// TIA Portal project "Project" (V15)

(* hardware
DEVICE "S7300/ET200M station_2"  S7-300 station
   slot 0: "Rail_0"  Rail  6ES7 390-1***0-0AA0
   slot 2: "PLC_2"  CPU 319-3 PN/DP  6ES7 318-3EL01-0AB0  V3.2
      slot 2: "DP interface_1"  DP
      slot 3: "PROFINET interface_1"  PN-IO
         slot 1: "Port_1"  Port
         slot 2: "Port_2"  Port
   slot 4: "DI 16/DO 16x24VDC/0.5A_1"  DI16/DO16 x 24V / 0.5A  6ES7 323-1BL00-0AA0
   slot 5: "DI 16/DO 16x24VDC/0.5A_2"  DI16/DO16 x 24V / 0.5A  6ES7 323-1BL00-0AA0
   slot 6: "DI 16/DO 16x24VDC/0.5A_3"  DI16/DO16 x 24V / 0.5A  6ES7 323-1BL00-0AA0
   slot 7: "DI 16/DO 16x24VDC/0.5A_4"  DI16/DO16 x 24V / 0.5A  6ES7 323-1BL00-0AA0
   slot 8: "DI 16/DO 16x24VDC/0.5A_5"  DI16/DO16 x 24V / 0.5A  6ES7 323-1BL00-0AA0
   slot 9: "DI 16/DO 16x24VDC/0.5A_6"  DI16/DO16 x 24V / 0.5A  6ES7 323-1BL00-0AA0
   slot 10: "DI 16/DO 16x24VDC/0.5A_7"  DI16/DO16 x 24V / 0.5A  6ES7 323-1BL00-0AA0
   slot 11: "DI 16/DO 16x24VDC/0.5A_8"  DI16/DO16 x 24V / 0.5A  6ES7 323-1BL00-0AA0
*)

// ===== PLC "PLC_2"  CPU 319-3 PN/DP =====

VAR_GLOBAL   // PLC tag table "All_Tags"
   "CCC1" AT %I10.0 : Bool;
   "CCC2" AT %I10.1 : Bool;
   "Tag_1" AT %M5.6 : Bool;
   "Tag_2" AT %M5.7 : Bool;
   "Tag_3" AT %M6.0 : Bool;
   "Tag_4" AT %M6.1 : Bool;
   "Tag_5" AT %M6.2 : Bool;
   "Tag_6" AT %M6.3 : Bool;
   "Tag_7" AT %M6.4 : Bool;
   "Tag_8" AT %M6.5 : Bool;
   "Tag_9" AT %M6.6 : Bool;
END_VAR

VAR_GLOBAL   // PLC tag table "base_feeding_station"
   "lid_detection" AT %I0.0 : Bool;
   "stop_beginning_lid_sensor" AT %I0.1 : Bool;
   "start_LID_feeding_convyer" AT %I0.2 : Bool;
   "LID_detected_grip" AT %I0.3 : Bool;
   "stop_LID_Feeding" AT %I0.4 : Bool;
   "LID_machining_entrance_sensor" AT %I0.5 : Bool;
   "base_Raw_counter_start" AT %I0.6 : Bool;
   "stop_base_begininning_convyr" AT %I0.7 : Bool;
   "base_gripper_detected" AT %I1.0 : Bool;
   "start_base_raw_feeding" AT %I1.1 : Bool;
   "stop_base_raw_feeding" AT %I1.2 : Bool;
   "stop_base_machining_convyr" AT %I1.3 : Bool;
   "lid_start_button" AT %I1.4 : Bool;
   "lid_stop_button" AT %I1.5 : Bool;
   "lid_emergency_button" AT %I1.6 : Bool;
   "base_start_button" AT %I1.7 : Bool;
   "base_stop_button" AT %I2.0 : Bool;
   "base_emergency" AT %I2.1 : Bool;
   "Lid_beginning_conveyr" AT %Q0.0 : Bool;
   "lid_feeding_conveyr" AT %Q0.1 : Bool;
   "Lid_pickup_x_axis" AT %Q0.3 : Bool;
   "lid_pickup_z_axis" AT %Q0.4 : Bool;
   "lid_sucction_gripper" AT %Q0.5 : Bool;
   "base_beginning_conveyr" AT %Q0.6 : Bool;
   "lid-machinning_conveyr" AT %Q0.2 : Bool;
   "base_raw_feeding_conveyr" AT %Q0.7 : Bool;
   "base_to_machinning_conveyr" AT %Q1.0 : Bool;
   "base_pickup_x_axis" AT %Q1.1 : Bool;
   "base_pickup_z_axis" AT %Q1.2 : Bool;
   "base_sucction_gripper" AT %Q1.3 : Bool;
   "base_start_button_1_light" AT %Q1.4 : Bool;
   "base_stop_button_1_light" AT %Q1.5 : Bool;
   "lid_start_light" AT %Q1.6 : Bool;
   "lid_stop_button_1_light" AT %Q1.7 : Bool;
   "base_raw_material" AT %Q2.0 : Bool;
   "lid_raw_emit" AT %Q2.1 : Bool;
   "state_of_start_base" AT %M0.0 : Bool;
   "state_of_start_LID" AT %M0.1 : Bool;
   "state_of_lid" AT %M0.2 : Bool;
   "dummy" AT %M0.3 : Bool;
   "To_emit_lid" AT %M0.4 : Bool;
   "item_ready_to_picked" AT %M0.5 : Bool;
   "movin_lid_z_mem" AT %M0.6 : Bool;
   "LID_moving_z_sensor" AT %I2.4 : Bool;
   "LID_moving_x_sensor" AT %I2.5 : Bool;
   "dummy(1)" AT %M0.7 : Bool;
   "dummy(2)" AT %M1.0 : Bool;
   "lid_belt_convyer_excess" AT %Q2.2 : Bool;
   "push_excess_blue_lid" AT %Q2.3 : Bool;
   "push_excess_green_lid" AT %Q2.4 : Bool;
   "Blue_vision_lid" AT %I2.6 : Bool;
   "green_vision_lid" AT %I2.7 : Bool;
   "front_blue_push_lid" AT %I3.0 : Bool;
   "back_blue_push_lid" AT %I3.1 : Bool;
   "front_green_push_lid" AT %I3.2 : Bool;
   "back_green_push_lid" AT %I3.3 : Bool;
   "into_cnc_lid_sensor" AT %I3.4 : Bool;
   "CNC_lid_empty" AT %M1.1 : Bool;
   "ONE_OBJECT_IN" AT %Q2.5 : Bool;
   "KEEP_DISTANCE" AT %Q2.6 : Bool;
   "ARE_WE_THERE_YET_BLUE_lid" AT %M1.2 : Bool;
   "ARE_WE_THERE_YET_GREEN_lid" AT %M1.3 : Bool;
   "LID_COUNTER_RESET_BUTTON_BLUE" AT %I3.5 : Bool;
   "TO_STORAGE_BLUE_CONVYER_lid" AT %Q2.7 : Bool;
   "TO_STORAGE_GREEN_CONVYER_lid" AT %Q3.0 : Bool;
   "TO_STORAGE_BLUE_SENSOR_lid" AT %I3.6 : Bool;
   "TO_STORAGE_GREEN_SENSOR_lid" AT %I3.7 : Bool;
   "LID_COUNTER_RESET_BUTTON_GREEN" AT %I4.0 : Bool;
   "GREEN_LID_PUSHER_SORTING(FRONT LIMIT)" AT %I4.1 : Bool;
   "GREEN_LID_PUSHER_SORTING(BACK LIMITT)" AT %I4.2 : Bool;
   "BLUE_LID_PUSHER_SORTING(FRONT LIMIT)" AT %I4.3 : Bool;
   "BLUE_LID_PUSHER_SORTING(BACK LIMIT)" AT %I4.4 : Bool;
   "BEGIN_SORTING_STATION_LIDS" AT %I4.5 : Bool;
   "BLUE_LID_VISION_SORTING" AT %I4.6 : Bool;
   "GREEN_LID_VISION_SORTING" AT %I4.7 : Bool;
   "SORTING_CONVYER_LID" AT %Q3.1 : Bool;
   "GREEN_LID_PUSHER_SORTING" AT %Q3.2 : Bool;
   "BLUE_LID_PUSHER_SORTING" AT %Q3.3 : Bool;
   "CNC_base_empty" AT %M2.5 : Bool;
   "to_emit_base" AT %M1.5 : Bool;
   "base_into_cnc" AT %I5.0 : Bool;
   "BASE_MOVE_X_SENSOR" AT %I5.1 : Bool;
   "BASE_MOVE_Z_SENSOR" AT %I5.2 : Bool;
   "DUMMY1" AT %M1.6 : Bool;
   "DUMMY2" AT %M1.7 : Bool;
   "DUMMY3" AT %M2.0 : Bool;
   "DUMMY4" AT %M2.1 : Bool;
   "DUMMY5" AT %M2.2 : Bool;
   "BASE_RAW_EXESS_CONV" AT %Q3.4 : Bool;
   "Are_we_there_base_raw_blue" AT %M2.3 : Bool;
   "Are_we_there_base_raw_green" AT %M2.4 : Bool;
   "base_raw_blue_exes_vision" AT %I5.3 : Bool;
   "base_raw_green_exes_vision" AT %I5.4 : Bool;
   "to_blue_base_raw_storage_sensor" AT %I5.5 : Bool;
   "to_green_base_raw_storage_sensor" AT %I5.6 : Bool;
   "push_ex_green_base raw(front)" AT %I5.7 : Bool;
   "push_ex_green_base raw (back)" AT %I6.0 : Bool;
   "pusher blue base raw (front)" AT %I6.1 : Bool;
   "pusher blue base raw (back)" AT %I6.2 : Bool;
   "is_base_exsist" AT %M1.4 : Bool;
   "Conv_sorting_set_base" AT %M2.6 : Bool;
   "BEGIN_SORTING_STATION_BASE_4" AT %Q5.3 : Bool;
END_VAR

VAR_GLOBAL   // PLC tag table "Assembly_tags"
   "Assembly green lid start" AT %I8.0 : Bool;
   "Assembly blue lid start" AT %I8.1 : Bool;
   "Assembly green base start" AT %I8.2 : Bool;
   "Assembly blue base start" AT %I8.3 : Bool;
   "G_lid in place" AT %I8.4 : Bool;
   "G_base in place" AT %I8.5 : Bool;
   "G_lid_clamped" AT %I8.6 : Bool;
   "G_base_clamped" AT %I8.7 : Bool;
   "G_part_leaving" AT %I9.0 : Bool;
   "G_item_detect" AT %I9.1 : Bool;
   "B_lid in place" AT %I9.2 : Bool;
   "B_base in place" AT %I9.3 : Bool;
   "B_lid_clamped" AT %I9.4 : Bool;
   "B_base_clamped" AT %I9.5 : Bool;
   "B_part_leaving" AT %I9.6 : Bool;
   "B_item_detect" AT %I9.7 : Bool;
   "G_Negative_Trig_1" AT %M4.0 : Bool;
   "G_Negative_Trig_2" AT %M4.1 : Bool;
   "G_Negative_Trig_3" AT %M4.2 : Bool;
   "move_green_lid_conv" AT %M4.3 : Bool;
   "move_green_base_conv" AT %M4.4 : Bool;
   "move_blue_lid_conv" AT %M4.5 : Bool;
   "move_blue_base_conv" AT %M4.6 : Bool;
   "B_Negative_Trig_1" AT %M4.7 : Bool;
   "B_Negative_Trig_2" AT %M5.0 : Bool;
   "B_Negative_Trig_3" AT %M5.1 : Bool;
   "G_Detected_Memory" AT %M5.2 : Bool;
   "G_Reset" AT %M5.3 : Bool;
   "B_Detected_Memory" AT %M5.4 : Bool;
   "B_Reset" AT %M5.5 : Bool;
   "G_Timer_1" AT %T0 : Timer;
   "G_Timer_2" AT %T1 : Timer;
   "G_Timer_3" AT %T2 : Timer;
   "B_Timer_1" AT %T3 : Timer;
   "B_Timer_2" AT %T4 : Timer;
   "B_Timer_3" AT %T5 : Timer;
   "G_lids_conv_1" AT %Q7.0 : Bool;
   "G_lids_conv_2" AT %Q7.1 : Bool;
   "G_lids_conv_3" AT %Q7.2 : Bool;
   "G_lids_conv_4" AT %Q7.3 : Bool;
   "G_lids_conv_5" AT %Q7.4 : Bool;
   "G_lids_conv_6" AT %Q7.5 : Bool;
   "G_lids_conv_7" AT %Q7.6 : Bool;
   "G_lids_conv_8" AT %Q7.7 : Bool;
   "B_lids_conv_1" AT %Q8.0 : Bool;
   "B_lids_conv_2" AT %Q8.1 : Bool;
   "B_lids_conv_3" AT %Q8.2 : Bool;
   "B_lids_conv_4" AT %Q8.3 : Bool;
   "G_base_conv_1" AT %Q8.4 : Bool;
   "G_base_conv_2" AT %Q8.5 : Bool;
   "G_base_conv_3" AT %Q8.6 : Bool;
   "G_base_conv_4" AT %Q8.7 : Bool;
   "G_base_conv_5" AT %Q9.0 : Bool;
   "G_base_conv_6" AT %Q9.1 : Bool;
   "B_base_conv_1" AT %Q9.2 : Bool;
   "B_base_conv_2" AT %Q9.3 : Bool;
   "B_base_conv_3" AT %Q9.4 : Bool;
   "B_base_conv_4" AT %Q9.5 : Bool;
   "G_clamp_lid" AT %Q9.6 : Bool;
   "G_clamp_base" AT %Q9.7 : Bool;
   "G_move Z" AT %Q10.0 : Bool;
   "G_grab" AT %Q10.1 : Bool;
   "G_move X" AT %Q10.2 : Bool;
   "G_pos.Raise_bases" AT %Q10.3 : Bool;
   "B_clamp_lid" AT %Q10.4 : Bool;
   "B_clamp_base" AT %Q10.5 : Bool;
   "B_move Z" AT %Q10.6 : Bool;
   "B_grab" AT %Q10.7 : Bool;
   "B_move X" AT %Q11.0 : Bool;
   "B_pos.Raise_bases" AT %Q11.1 : Bool;
END_VAR

VAR_GLOBAL   // PLC tag table "Default tag table"
   "MachineCenter1_lid_start" AT %Q3.5 : Bool;
   "MachineCenter1_lid_produceLids" AT %Q3.6 : Bool;
   "push_excess_blue_base" AT %Q3.7 : Bool;
   "push_excess_green_base" AT %Q4.0 : Bool;
   "base_COUNTER_RESET_BUTTON_BLUE" AT %I6.3 : Bool;
   "base_COUNTER_RESET_BUTTON_GREEN" AT %I6.4 : Bool;
   "base_raw_excess_blue" AT %Q4.1 : Bool;
   "base_raw_excess_green" AT %Q4.2 : Bool;
   "base_vision_raw_execess_sensor_green" AT %I6.5 : Bool;
   "base_vision_raw_execess_sensor_blue" AT %I6.6 : Bool;
   "MachineCenter2_base_start" AT %Q4.3 : Bool;
   "Stop_blade4" AT %Q4.4 : Bool;
   "Stop_blade5" AT %Q4.5 : Bool;
   "MACHINE1_BUSY" AT %I6.7 : Bool;
   "BEGIN_SORTING_STATION_BASE_SENSOR" AT %I7.0 : Bool;
   "BEGIN_SORTING_STATION_BASE_1" AT %Q4.6 : Bool;
   "BEGIN_SORTING_STATION_BASE_2" AT %Q4.7 : Bool;
   "BEGIN_SORTING_STATION_BASE_3" AT %Q5.0 : Bool;
   "Green_base_sorting_vision" AT %I7.1 : Bool;
   "Blue_base_sorting_vision" AT %I7.2 : Bool;
   "Pusher_green_base (Front Limit)" AT %I7.3 : Bool;
   "Pusher_green_base (Back Limit)" AT %I7.4 : Bool;
   "Pusher_blue_base (Front Limit)" AT %I7.5 : Bool;
   "Pusher_blue_base (Back Limit)" AT %I7.6 : Bool;
   "Pusher_blue_base_sorter" AT %Q5.2 : Bool;
   "Pusher_green_base_sorter" AT %Q5.1 : Bool;
   "Conv_sorting_set_lid" AT %M2.7 : Bool;
   "Emit_set_lid" AT %M3.0 : Bool;
   "Emit_set_base" AT %M3.1 : Bool;
   "Blue count" AT %MW4 : Int;
   "excess blue lid raw led light" AT %Q5.4 : Bool;
   "excess green lid raw led light" AT %Q5.5 : Bool;
   "excess blue base raw led light" AT %Q5.6 : Bool;
   "excess green base raw led light" AT %Q5.7 : Bool;
   "blue lid sorting light" AT %Q6.0 : Bool;
   "green lid sorting light" AT %Q6.1 : Bool;
   "blue base sorting light" AT %Q6.2 : Bool;
   "green base sorting light" AT %Q6.3 : Bool;
   "Green_Lid_conv_timer" AT %T6 : Timer;
   "Blue_Lid_conv_timer" AT %T7 : Timer;
   "Green_Base_conv_timer" AT %T8 : Timer;
   "Blue_Base_conv_timer" AT %T9 : Timer;
END_VAR

DATA_BLOCK "Data_block_1ddd"   // DB3
{ S7_Optimized_Access := 'FALSE' }
VERSION : 0.1
BEGIN
END_DATA_BLOCK

DATA_BLOCK "PICK_UP_LID_ROBOT_DB"   // DB11
{ S7_Optimized_Access := 'FALSE' }
VERSION : 0.1
// stored: InstanceOfName PICK_UP_LID_ROBOT
"PICK_UP_LID_ROBOT"
BEGIN
END_DATA_BLOCK

DATA_BLOCK "LID_SORTING_STATION_DB"   // DB12
{ S7_Optimized_Access := 'FALSE' }
VERSION : 0.1
// stored: InstanceOfName LID_SORTING_STATION
"LID_SORTING_STATION"
BEGIN
END_DATA_BLOCK

DATA_BLOCK "LID PRODUCTION_DB"   // DB13
{ S7_Optimized_Access := 'FALSE' }
VERSION : 0.1
// stored: InstanceOfName LID PRODUCTION
"LID PRODUCTION"
BEGIN
END_DATA_BLOCK

DATA_BLOCK "LID_execess_remove_station_DB"   // DB14
{ S7_Optimized_Access := 'FALSE' }
VERSION : 0.1
// stored: InstanceOfName LID_execess_remove_station
"LID_execess_remove_station"
BEGIN
END_DATA_BLOCK

DATA_BLOCK "base_production_fb_DB"   // DB17
{ S7_Optimized_Access := 'FALSE' }
VERSION : 0.1
// stored: InstanceOfName base_production_fb
"base_production_fb"
BEGIN
END_DATA_BLOCK

DATA_BLOCK "PICK_UP_BASE_ROBOT_DB"   // DB19
{ S7_Optimized_Access := 'FALSE' }
VERSION : 0.1
// stored: InstanceOfName PICK_UP_BASE_ROBOT
"PICK_UP_BASE_ROBOT"
BEGIN
END_DATA_BLOCK

DATA_BLOCK "PICK_UP_BASE_ROBOT_DB_1"   // DB20
{ S7_Optimized_Access := 'FALSE' }
VERSION : 0.1
// stored: InstanceOfName PICK_UP_BASE_ROBOT
"PICK_UP_BASE_ROBOT"
BEGIN
END_DATA_BLOCK

DATA_BLOCK "BASE_execess_remove_station_DB"   // DB26
{ S7_Optimized_Access := 'FALSE' }
VERSION : 0.1
// stored: InstanceOfName BASE_execess_remove_station
"BASE_execess_remove_station"
BEGIN
END_DATA_BLOCK

DATA_BLOCK "A_COUNTER_DB_1"   // DB27
{ S7_Optimized_Access := 'FALSE' }
VERSION : 0.1
// stored: InstanceOfName A_COUNTER
"A_COUNTER"
BEGIN
END_DATA_BLOCK

DATA_BLOCK "BASE_SORTING_STATION_DB"   // DB28
{ S7_Optimized_Access := 'FALSE' }
VERSION : 0.1
// stored: InstanceOfName BASE_SORTING_STATION
"BASE_SORTING_STATION"
BEGIN
END_DATA_BLOCK

DATA_BLOCK "Block_1_DB"   // DB30
{ S7_Optimized_Access := 'FALSE' }
VERSION : 0.1
// stored: InstanceOfName A_COUNTER
"A_COUNTER"
BEGIN
END_DATA_BLOCK

DATA_BLOCK "Assembly_conv_DB"   // DB31
{ S7_Optimized_Access := 'FALSE' }
VERSION : 0.1
// stored: InstanceOfName Assembly_conv
"Assembly_conv"
BEGIN
END_DATA_BLOCK

DATA_BLOCK "Assembly_Blue_DB"   // DB32
{ S7_Optimized_Access := 'FALSE' }
VERSION : 0.1
// stored: InstanceOfName Assembly_Blue
"Assembly_Blue"
BEGIN
END_DATA_BLOCK

DATA_BLOCK "Assembly_Green_DB"   // DB33
{ S7_Optimized_Access := 'FALSE' }
VERSION : 0.1
// stored: InstanceOfName Assembly_Green
"Assembly_Green"
BEGIN
END_DATA_BLOCK

DATA_BLOCK "Assembly_Emergency_DB_1"   // DB34
{ S7_Optimized_Access := 'FALSE' }
VERSION : 0.1
// stored: InstanceOfName Assembly_Emergency
"Assembly_Emergency"
BEGIN
END_DATA_BLOCK

DATA_BLOCK "Assembly_Emergency_DB"   // DB35
{ S7_Optimized_Access := 'FALSE' }
VERSION : 0.1
// stored: InstanceOfName Assembly_Emergency
"Assembly_Emergency"
BEGIN
END_DATA_BLOCK

DATA_BLOCK "A_COUNTER_DB"   // DB36
{ S7_Optimized_Access := 'FALSE' }
VERSION : 0.1
// stored: InstanceOfName A_COUNTER
"A_COUNTER"
BEGIN
END_DATA_BLOCK

FUNCTION_BLOCK "PICK_UP_LID_ROBOT"   // FB1, LAD
{ S7_Optimized_Access := 'FALSE' }
VERSION : 0.1
   VAR_TEMP   // added for the SCL form of the ladder/FBD networks
      _w1 : Bool;
   END_VAR
BEGIN

REGION Network 1: LID_PICKUP_ROBOT_LOWERING_Z_AXIS
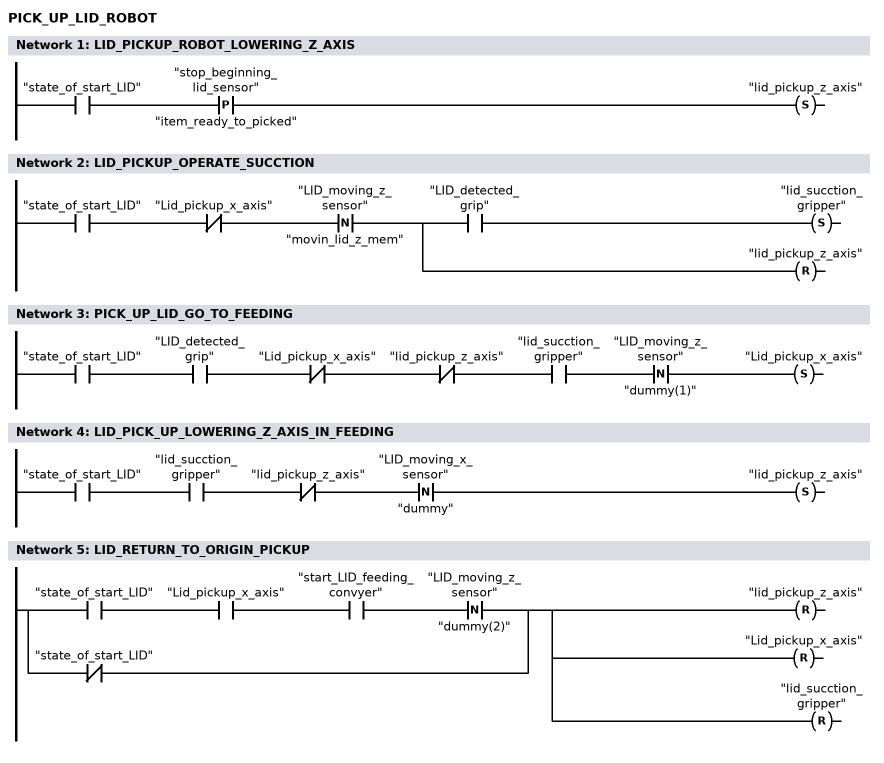
   RUNG wire#powerrail
      Contact( "state_of_start_LID" )
      P_Contact(operand := "stop_beginning_lid_sensor", bit := "item_ready_to_picked")
      S_Coil( "lid_pickup_z_axis" )
   END_RUNG
   // the same network as SCL:
   #_w1 := "state_of_start_LID" AND "stop_beginning_lid_sensor" AND NOT "item_ready_to_picked";   // rising edge of "stop_beginning_lid_sensor"
   "item_ready_to_picked" := "stop_beginning_lid_sensor";
   IF #_w1 THEN "lid_pickup_z_axis" := TRUE; END_IF;
END_REGION

REGION Network 2: LID_PICKUP_OPERATE_SUCCTION
   RUNG wire#powerrail
      Contact( "state_of_start_LID" )
      I_Contact( "Lid_pickup_x_axis" )
      N_Contact(operand := "LID_moving_z_sensor", bit := "movin_lid_z_mem")
      wire#w1
      Contact( "LID_detected_grip" )
      S_Coil( "lid_sucction_gripper" )
   END_RUNG
   RUNG wire#w1
      R_Coil( "lid_pickup_z_axis" )
   END_RUNG
   // the same network as SCL:
   #_w1 := "state_of_start_LID" AND NOT "Lid_pickup_x_axis" AND NOT "LID_moving_z_sensor" AND "movin_lid_z_mem";   // falling edge of "LID_moving_z_sensor"
   "movin_lid_z_mem" := "LID_moving_z_sensor";
   IF #_w1 AND "LID_detected_grip" THEN "lid_sucction_gripper" := TRUE; END_IF;
   IF #_w1 THEN "lid_pickup_z_axis" := FALSE; END_IF;
END_REGION

REGION Network 3: PICK_UP_LID_GO_TO_FEEDING
   RUNG wire#powerrail
      Contact( "state_of_start_LID" )
      Contact( "LID_detected_grip" )
      I_Contact( "Lid_pickup_x_axis" )
      I_Contact( "lid_pickup_z_axis" )
      Contact( "lid_sucction_gripper" )
      N_Contact(operand := "LID_moving_z_sensor", bit := "dummy(1)")
      S_Coil( "Lid_pickup_x_axis" )
   END_RUNG
   // the same network as SCL:
   #_w1 := "state_of_start_LID" AND "LID_detected_grip" AND NOT "Lid_pickup_x_axis" AND NOT "lid_pickup_z_axis" AND "lid_sucction_gripper" AND NOT "LID_moving_z_sensor" AND "dummy(1)";   // falling edge of "LID_moving_z_sensor"
   "dummy(1)" := "LID_moving_z_sensor";
   IF #_w1 THEN "Lid_pickup_x_axis" := TRUE; END_IF;
END_REGION

REGION Network 4: LID_PICK_UP_LOWERING_Z_AXIS_IN_FEEDING
   RUNG wire#powerrail
      Contact( "state_of_start_LID" )
      Contact( "lid_sucction_gripper" )
      I_Contact( "lid_pickup_z_axis" )
      N_Contact(operand := "LID_moving_x_sensor", bit := "dummy")
      S_Coil( "lid_pickup_z_axis" )
   END_RUNG
   // the same network as SCL:
   #_w1 := "state_of_start_LID" AND "lid_sucction_gripper" AND NOT "lid_pickup_z_axis" AND NOT "LID_moving_x_sensor" AND "dummy";   // falling edge of "LID_moving_x_sensor"
   "dummy" := "LID_moving_x_sensor";
   IF #_w1 THEN "lid_pickup_z_axis" := TRUE; END_IF;
END_REGION

REGION Network 5: LID_RETURN_TO_ORIGIN_PICKUP
   RUNG wire#powerrail
      Contact( "state_of_start_LID" )
      Contact( "Lid_pickup_x_axis" )
      Contact( "start_LID_feeding_convyer" )
      N_Contact(operand := "LID_moving_z_sensor", bit := "dummy(2)")
      wire#w1
      R_Coil( "lid_pickup_z_axis" )
   END_RUNG
   RUNG wire#powerrail
      I_Contact( "state_of_start_LID" )
   END_RUNG wire#w1
   RUNG wire#w1
      R_Coil( "Lid_pickup_x_axis" )
   END_RUNG
   RUNG wire#w1
      R_Coil( "lid_sucction_gripper" )
   END_RUNG
   // the same network as SCL:
   #_w1 := "state_of_start_LID" AND "Lid_pickup_x_axis" AND "start_LID_feeding_convyer" AND NOT "LID_moving_z_sensor" AND "dummy(2)";   // falling edge of "LID_moving_z_sensor"
   "dummy(2)" := "LID_moving_z_sensor";
   IF #_w1 OR NOT "state_of_start_LID" THEN
       "lid_pickup_z_axis" := FALSE;
       "Lid_pickup_x_axis" := FALSE;
       "lid_sucction_gripper" := FALSE;
   END_IF;
END_REGION
END_FUNCTION_BLOCK

FUNCTION_BLOCK "LID PRODUCTION"   // FB2, LAD
{ S7_Optimized_Access := 'FALSE' }
VERSION : 0.1
BEGIN

REGION Network 1: LID STARTING HANDLE
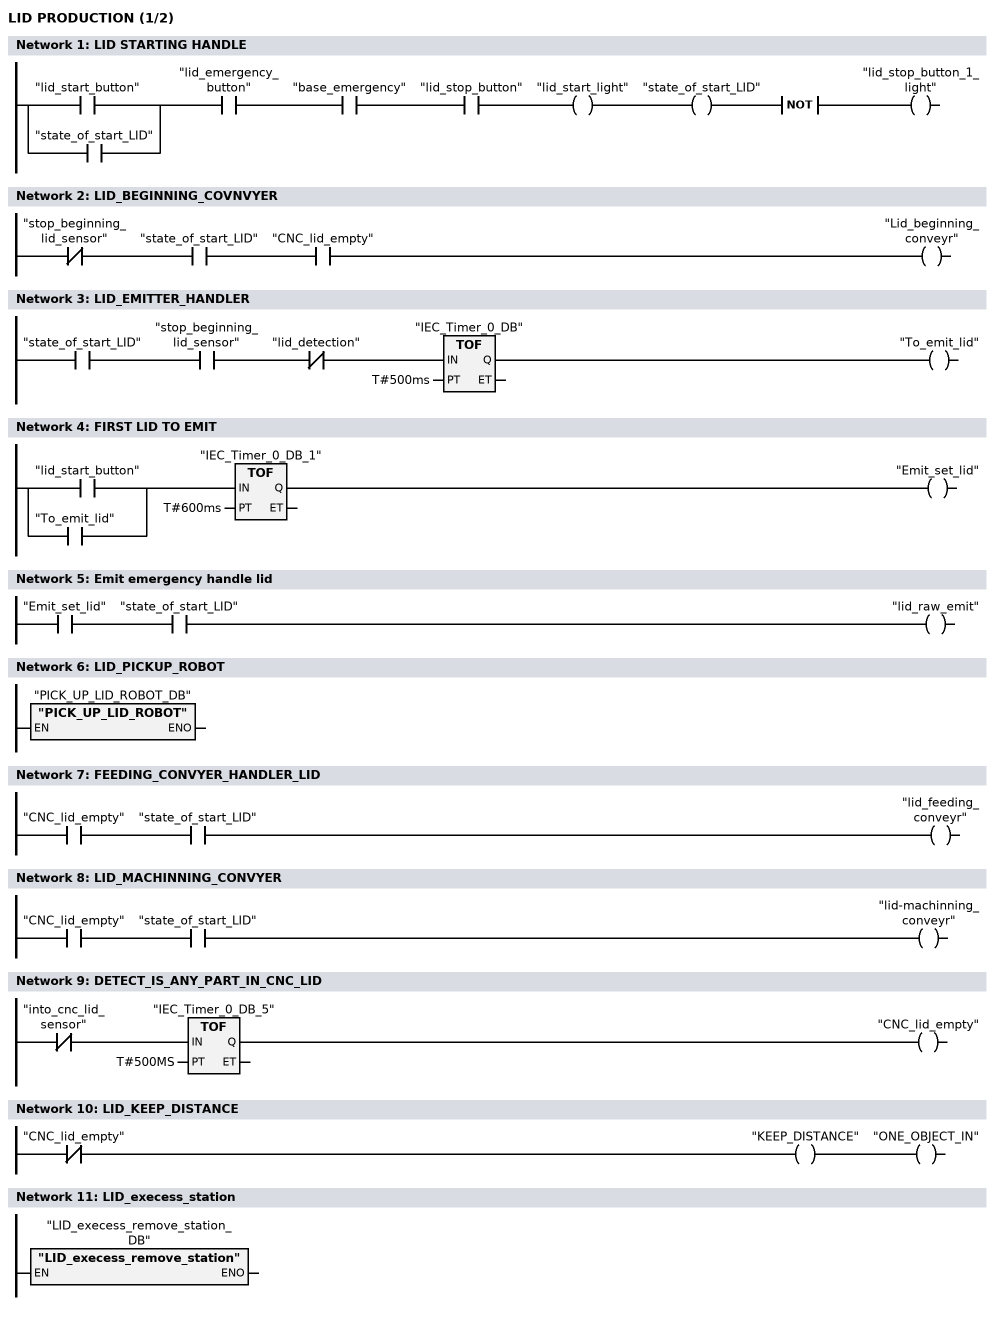
   RUNG wire#powerrail
      Contact( "lid_start_button" )
      wire#w1
      Contact( "lid_emergency_button" )
      Contact( "base_emergency" )
      Contact( "lid_stop_button" )
      Coil( "lid_start_light" )
      Coil( "state_of_start_LID" )
      Not()
      Coil( "lid_stop_button_1_light" )
   END_RUNG
   RUNG wire#powerrail
      Contact( "state_of_start_LID" )
   END_RUNG wire#w1
   // the same network as SCL:
   "lid_start_light" := ("lid_start_button" OR "state_of_start_LID") AND "lid_emergency_button" AND "base_emergency" AND "lid_stop_button";
   "state_of_start_LID" := "lid_start_light";
   "lid_stop_button_1_light" := NOT "lid_start_light";
END_REGION

REGION Network 2: LID_BEGINNING_COVNVYER
   RUNG wire#powerrail
      I_Contact( "stop_beginning_lid_sensor" )
      Contact( "state_of_start_LID" )
      Contact( "CNC_lid_empty" )
      Coil( "Lid_beginning_conveyr" )
   END_RUNG
   // the same network as SCL:
   "Lid_beginning_conveyr" := NOT "stop_beginning_lid_sensor" AND "state_of_start_LID" AND "CNC_lid_empty";
END_REGION

REGION Network 3: LID_EMITTER_HANDLER
   "IEC_Timer_0_DB".TOF(IN := "state_of_start_LID" AND "stop_beginning_lid_sensor" AND NOT "lid_detection",
                        PT := T#500ms);
   "To_emit_lid" := "IEC_Timer_0_DB".Q;
END_REGION

REGION Network 4: FIRST LID TO EMIT
   "IEC_Timer_0_DB_1".TOF(IN := "lid_start_button" OR "To_emit_lid", PT := T#600ms);
   "Emit_set_lid" := "IEC_Timer_0_DB_1".Q;
END_REGION

REGION Network 5: Emit emergency handle lid
   RUNG wire#powerrail
      Contact( "Emit_set_lid" )
      Contact( "state_of_start_LID" )
      Coil( "lid_raw_emit" )
   END_RUNG
   // the same network as SCL:
   "lid_raw_emit" := "Emit_set_lid" AND "state_of_start_LID";
END_REGION

REGION Network 6: LID_PICKUP_ROBOT
   RUNG wire#powerrail
      "PICK_UP_LID_ROBOT_DB"()
   END_RUNG
   // the same network as SCL:
   "PICK_UP_LID_ROBOT_DB"();   // "PICK_UP_LID_ROBOT"
END_REGION

REGION Network 7: FEEDING_CONVYER_HANDLER_LID
   RUNG wire#powerrail
      Contact( "CNC_lid_empty" )
      Contact( "state_of_start_LID" )
      Coil( "lid_feeding_conveyr" )
   END_RUNG
   // the same network as SCL:
   "lid_feeding_conveyr" := "CNC_lid_empty" AND "state_of_start_LID";
END_REGION

REGION Network 8: LID_MACHINNING_CONVYER
   RUNG wire#powerrail
      Contact( "CNC_lid_empty" )
      Contact( "state_of_start_LID" )
      Coil( "lid-machinning_conveyr" )
   END_RUNG
   // the same network as SCL:
   "lid-machinning_conveyr" := "CNC_lid_empty" AND "state_of_start_LID";
END_REGION

REGION Network 9: DETECT_IS_ANY_PART_IN_CNC_LID
   "IEC_Timer_0_DB_5".TOF(IN := NOT "into_cnc_lid_sensor", PT := T#500MS);
   "CNC_lid_empty" := "IEC_Timer_0_DB_5".Q;
END_REGION

REGION Network 10: LID_KEEP_DISTANCE
   RUNG wire#powerrail
      I_Contact( "CNC_lid_empty" )
      Coil( "KEEP_DISTANCE" )
      Coil( "ONE_OBJECT_IN" )
   END_RUNG
   // the same network as SCL:
   "KEEP_DISTANCE" := NOT "CNC_lid_empty";
   "ONE_OBJECT_IN" := NOT "CNC_lid_empty";
END_REGION

REGION Network 11: LID_execess_station
   RUNG wire#powerrail
      "LID_execess_remove_station_DB"()
   END_RUNG
   // the same network as SCL:
   "LID_execess_remove_station_DB"();   // "LID_execess_remove_station"
END_REGION

REGION Network 12: CNC
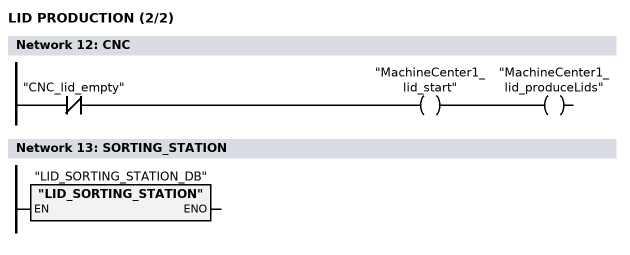
   RUNG wire#powerrail
      I_Contact( "CNC_lid_empty" )
      Coil( "MachineCenter1_lid_start" )
      Coil( "MachineCenter1_lid_produceLids" )
   END_RUNG
   // the same network as SCL:
   "MachineCenter1_lid_start" := NOT "CNC_lid_empty";
   "MachineCenter1_lid_produceLids" := NOT "CNC_lid_empty";
END_REGION

REGION Network 13: SORTING_STATION
   RUNG wire#powerrail
      "LID_SORTING_STATION_DB"()
   END_RUNG
   // the same network as SCL:
   "LID_SORTING_STATION_DB"();   // "LID_SORTING_STATION"
END_REGION
END_FUNCTION_BLOCK

FUNCTION_BLOCK "LID_SORTING_STATION"   // FB3, LAD
{ S7_Optimized_Access := 'FALSE' }
VERSION : 0.1
BEGIN

REGION Network 1: BEGIN SORTING CONVYER
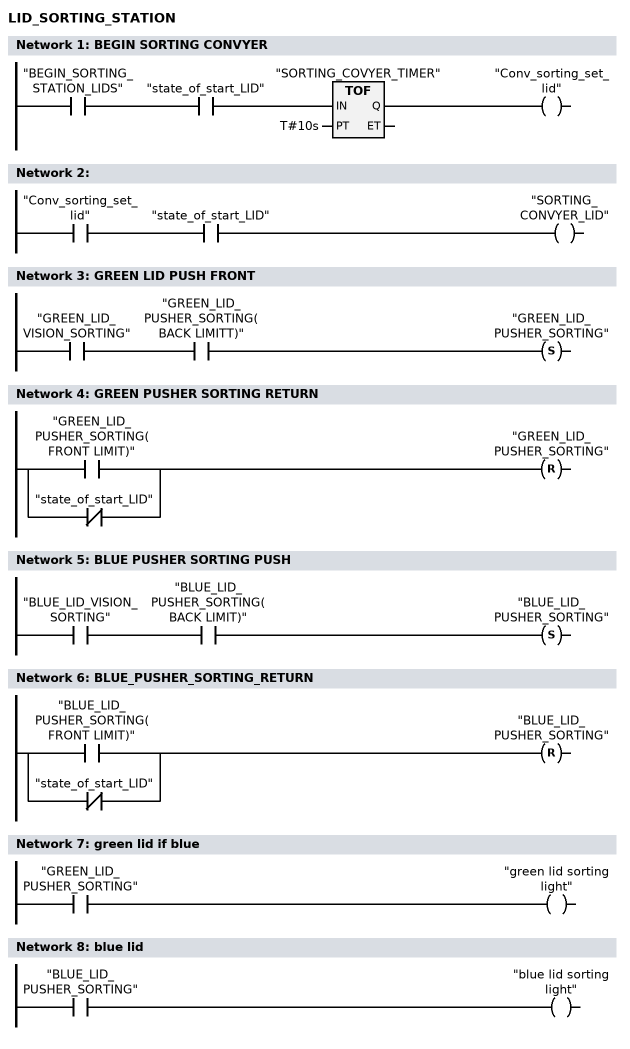
   "SORTING_COVYER_TIMER".TOF(IN := "BEGIN_SORTING_STATION_LIDS" AND "state_of_start_LID", PT := T#10s);
   "Conv_sorting_set_lid" := "SORTING_COVYER_TIMER".Q;
END_REGION

REGION Network 2
   RUNG wire#powerrail
      Contact( "Conv_sorting_set_lid" )
      Contact( "state_of_start_LID" )
      Coil( "SORTING_CONVYER_LID" )
   END_RUNG
   // the same network as SCL:
   "SORTING_CONVYER_LID" := "Conv_sorting_set_lid" AND "state_of_start_LID";
END_REGION

REGION Network 3: GREEN LID PUSH FRONT
   RUNG wire#powerrail
      Contact( "GREEN_LID_VISION_SORTING" )
      Contact( "GREEN_LID_PUSHER_SORTING(BACK LIMITT)" )
      S_Coil( "GREEN_LID_PUSHER_SORTING" )
   END_RUNG
   // the same network as SCL:
   IF "GREEN_LID_VISION_SORTING" AND "GREEN_LID_PUSHER_SORTING(BACK LIMITT)" THEN
       "GREEN_LID_PUSHER_SORTING" := TRUE;
   END_IF;
END_REGION

REGION Network 4: GREEN PUSHER SORTING RETURN
   RUNG wire#powerrail
      Contact( "GREEN_LID_PUSHER_SORTING(FRONT LIMIT)" )
      wire#w1
      R_Coil( "GREEN_LID_PUSHER_SORTING" )
   END_RUNG
   RUNG wire#powerrail
      I_Contact( "state_of_start_LID" )
   END_RUNG wire#w1
   // the same network as SCL:
   IF "GREEN_LID_PUSHER_SORTING(FRONT LIMIT)" OR NOT "state_of_start_LID" THEN
       "GREEN_LID_PUSHER_SORTING" := FALSE;
   END_IF;
END_REGION

REGION Network 5: BLUE PUSHER SORTING PUSH
   RUNG wire#powerrail
      Contact( "BLUE_LID_VISION_SORTING" )
      Contact( "BLUE_LID_PUSHER_SORTING(BACK LIMIT)" )
      S_Coil( "BLUE_LID_PUSHER_SORTING" )
   END_RUNG
   // the same network as SCL:
   IF "BLUE_LID_VISION_SORTING" AND "BLUE_LID_PUSHER_SORTING(BACK LIMIT)" THEN
       "BLUE_LID_PUSHER_SORTING" := TRUE;
   END_IF;
END_REGION

REGION Network 6: BLUE_PUSHER_SORTING_RETURN
   RUNG wire#powerrail
      Contact( "BLUE_LID_PUSHER_SORTING(FRONT LIMIT)" )
      wire#w1
      R_Coil( "BLUE_LID_PUSHER_SORTING" )
   END_RUNG
   RUNG wire#powerrail
      I_Contact( "state_of_start_LID" )
   END_RUNG wire#w1
   // the same network as SCL:
   IF "BLUE_LID_PUSHER_SORTING(FRONT LIMIT)" OR NOT "state_of_start_LID" THEN
       "BLUE_LID_PUSHER_SORTING" := FALSE;
   END_IF;
END_REGION

REGION Network 7: green lid if blue
   RUNG wire#powerrail
      Contact( "GREEN_LID_PUSHER_SORTING" )
      Coil( "green lid sorting light" )
   END_RUNG
   // the same network as SCL:
   "green lid sorting light" := "GREEN_LID_PUSHER_SORTING";
END_REGION

REGION Network 8: blue lid
   RUNG wire#powerrail
      Contact( "BLUE_LID_PUSHER_SORTING" )
      Coil( "blue lid sorting light" )
   END_RUNG
   // the same network as SCL:
   "blue lid sorting light" := "BLUE_LID_PUSHER_SORTING";
END_REGION
END_FUNCTION_BLOCK

FUNCTION_BLOCK "LID_execess_remove_station"   // FB4, LAD
{ S7_Optimized_Access := 'FALSE' }
VERSION : 0.1
   VAR_TEMP   // added for the SCL form of the ladder/FBD networks
      _w1 : Bool;
   END_VAR
BEGIN

REGION Network 1: LID_BELT_EXECESS_CONVYR_HANDLER
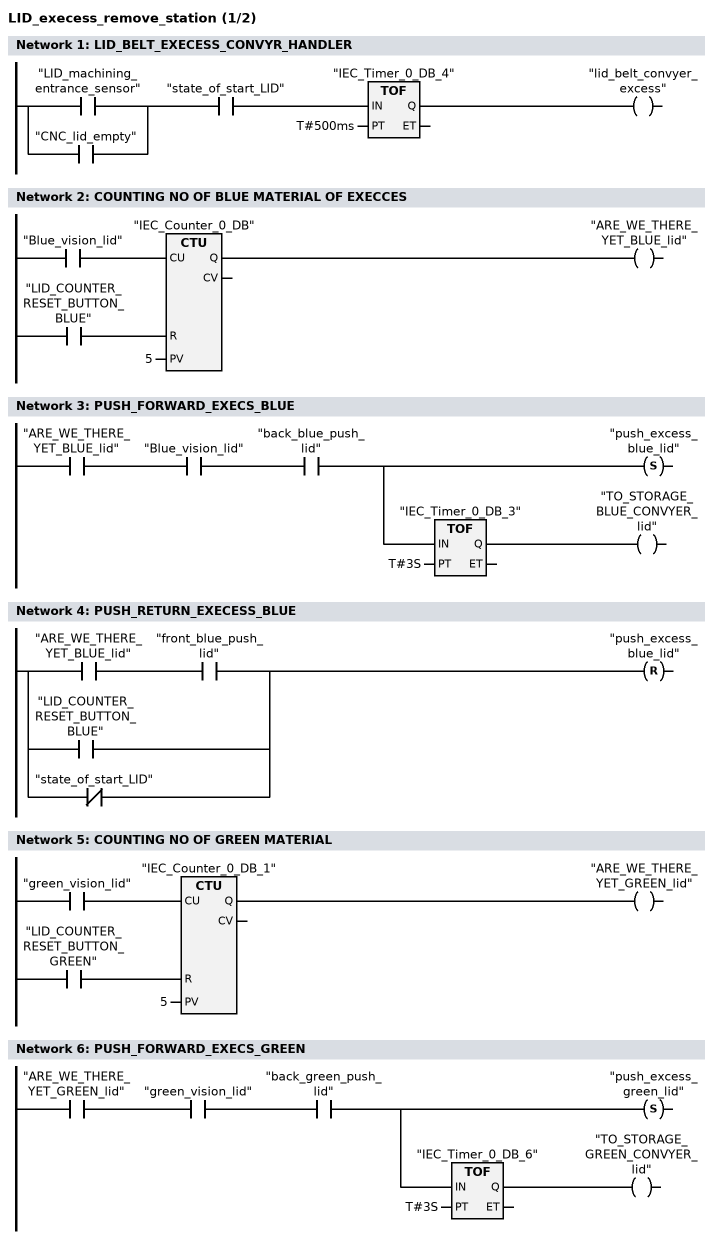
   "IEC_Timer_0_DB_4".TOF(IN := ("LID_machining_entrance_sensor" OR "CNC_lid_empty") AND "state_of_start_LID",
                          PT := T#500ms);
   "lid_belt_convyer_excess" := "IEC_Timer_0_DB_4".Q;
END_REGION

REGION Network 2: COUNTING NO OF BLUE MATERIAL OF EXECCES
   "IEC_Counter_0_DB".CTU(CU := "Blue_vision_lid", R := "LID_COUNTER_RESET_BUTTON_BLUE", PV := 5);
   "ARE_WE_THERE_YET_BLUE_lid" := "IEC_Counter_0_DB".Q;
END_REGION

REGION Network 3: PUSH_FORWARD_EXECS_BLUE
   #_w1 := "ARE_WE_THERE_YET_BLUE_lid" AND "Blue_vision_lid" AND "back_blue_push_lid";
   IF #_w1 THEN "push_excess_blue_lid" := TRUE; END_IF;
   "IEC_Timer_0_DB_3".TOF(IN := #_w1, PT := T#3S);
   "TO_STORAGE_BLUE_CONVYER_lid" := "IEC_Timer_0_DB_3".Q;
END_REGION

REGION Network 4: PUSH_RETURN_EXECESS_BLUE
   RUNG wire#powerrail
      Contact( "ARE_WE_THERE_YET_BLUE_lid" )
      Contact( "front_blue_push_lid" )
      wire#w1
      R_Coil( "push_excess_blue_lid" )
   END_RUNG
   RUNG wire#powerrail
      Contact( "LID_COUNTER_RESET_BUTTON_BLUE" )
   END_RUNG wire#w1
   RUNG wire#powerrail
      I_Contact( "state_of_start_LID" )
   END_RUNG wire#w1
   // the same network as SCL:
   IF ("ARE_WE_THERE_YET_BLUE_lid" AND "front_blue_push_lid") OR "LID_COUNTER_RESET_BUTTON_BLUE" OR NOT "state_of_start_LID" THEN
       "push_excess_blue_lid" := FALSE;
   END_IF;
END_REGION

REGION Network 5: COUNTING NO OF GREEN MATERIAL
   "IEC_Counter_0_DB_1".CTU(CU := "green_vision_lid", R := "LID_COUNTER_RESET_BUTTON_GREEN", PV := 5);
   "ARE_WE_THERE_YET_GREEN_lid" := "IEC_Counter_0_DB_1".Q;
END_REGION

REGION Network 6: PUSH_FORWARD_EXECS_GREEN
   #_w1 := "ARE_WE_THERE_YET_GREEN_lid" AND "green_vision_lid" AND "back_green_push_lid";
   IF #_w1 THEN "push_excess_green_lid" := TRUE; END_IF;
   "IEC_Timer_0_DB_6".TOF(IN := #_w1, PT := T#3S);
   "TO_STORAGE_GREEN_CONVYER_lid" := "IEC_Timer_0_DB_6".Q;
END_REGION

REGION Network 7: PUSH_RETURN_GREEN
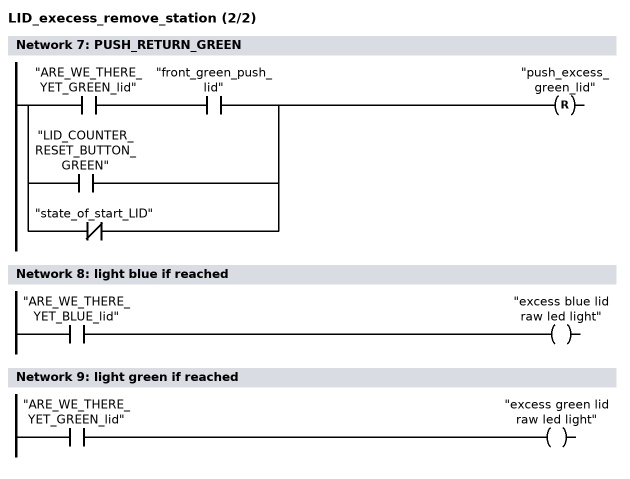
   RUNG wire#powerrail
      Contact( "ARE_WE_THERE_YET_GREEN_lid" )
      Contact( "front_green_push_lid" )
      wire#w1
      R_Coil( "push_excess_green_lid" )
   END_RUNG
   RUNG wire#powerrail
      Contact( "LID_COUNTER_RESET_BUTTON_GREEN" )
   END_RUNG wire#w1
   RUNG wire#powerrail
      I_Contact( "state_of_start_LID" )
   END_RUNG wire#w1
   // the same network as SCL:
   IF ("ARE_WE_THERE_YET_GREEN_lid" AND "front_green_push_lid") OR "LID_COUNTER_RESET_BUTTON_GREEN" OR NOT "state_of_start_LID" THEN
       "push_excess_green_lid" := FALSE;
   END_IF;
END_REGION

REGION Network 8: light blue if reached
   RUNG wire#powerrail
      Contact( "ARE_WE_THERE_YET_BLUE_lid" )
      Coil( "excess blue lid raw led light" )
   END_RUNG
   // the same network as SCL:
   "excess blue lid raw led light" := "ARE_WE_THERE_YET_BLUE_lid";
END_REGION

REGION Network 9: light green if reached
   RUNG wire#powerrail
      Contact( "ARE_WE_THERE_YET_GREEN_lid" )
      Coil( "excess green lid raw led light" )
   END_RUNG
   // the same network as SCL:
   "excess green lid raw led light" := "ARE_WE_THERE_YET_GREEN_lid";
END_REGION
END_FUNCTION_BLOCK

FUNCTION_BLOCK "base_production_fb"   // FB5, LAD
{ S7_Optimized_Access := 'FALSE' }
VERSION : 0.1
BEGIN

REGION Network 1: base_production_station
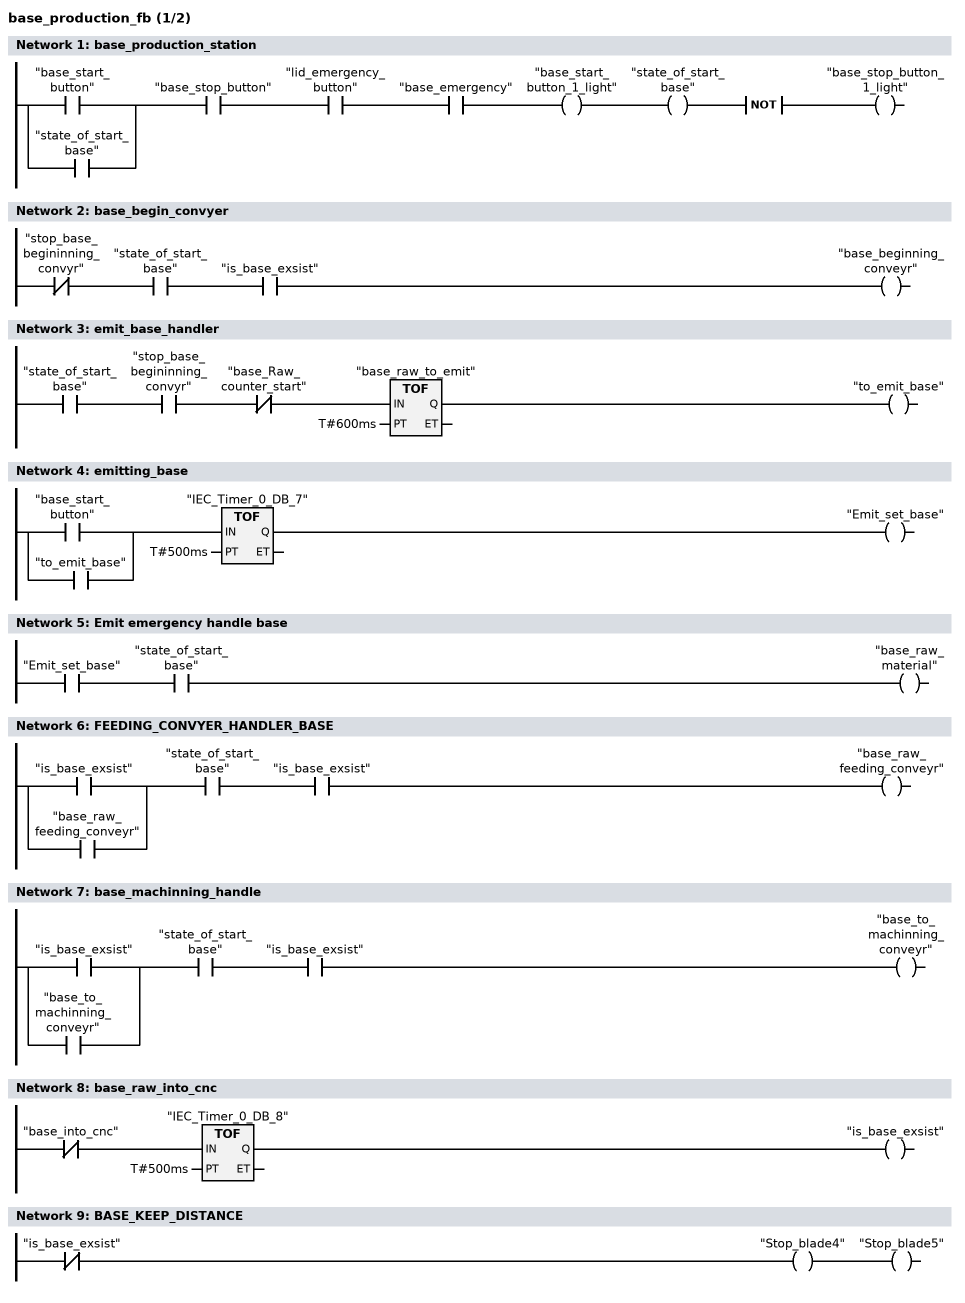
   RUNG wire#powerrail
      Contact( "base_start_button" )
      wire#w1
      Contact( "base_stop_button" )
      Contact( "lid_emergency_button" )
      Contact( "base_emergency" )
      Coil( "base_start_button_1_light" )
      Coil( "state_of_start_base" )
      Not()
      Coil( "base_stop_button_1_light" )
   END_RUNG
   RUNG wire#powerrail
      Contact( "state_of_start_base" )
   END_RUNG wire#w1
   // the same network as SCL:
   "base_start_button_1_light" := ("base_start_button" OR "state_of_start_base") AND "base_stop_button" AND "lid_emergency_button" AND "base_emergency";
   "state_of_start_base" := "base_start_button_1_light";
   "base_stop_button_1_light" := NOT "base_start_button_1_light";
END_REGION

REGION Network 2: base_begin_convyer
   RUNG wire#powerrail
      I_Contact( "stop_base_begininning_convyr" )
      Contact( "state_of_start_base" )
      Contact( "is_base_exsist" )
      Coil( "base_beginning_conveyr" )
   END_RUNG
   // the same network as SCL:
   "base_beginning_conveyr" := NOT "stop_base_begininning_convyr" AND "state_of_start_base" AND "is_base_exsist";
END_REGION

REGION Network 3: emit_base_handler
   "base_raw_to_emit".TOF(IN := "state_of_start_base" AND "stop_base_begininning_convyr" AND NOT "base_Raw_counter_start",
                          PT := T#600ms);
   "to_emit_base" := "base_raw_to_emit".Q;
END_REGION

REGION Network 4: emitting_base
   "IEC_Timer_0_DB_7".TOF(IN := "base_start_button" OR "to_emit_base", PT := T#500ms);
   "Emit_set_base" := "IEC_Timer_0_DB_7".Q;
END_REGION

REGION Network 5: Emit emergency handle base
   RUNG wire#powerrail
      Contact( "Emit_set_base" )
      Contact( "state_of_start_base" )
      Coil( "base_raw_material" )
   END_RUNG
   // the same network as SCL:
   "base_raw_material" := "Emit_set_base" AND "state_of_start_base";
END_REGION

REGION Network 6: FEEDING_CONVYER_HANDLER_BASE
   RUNG wire#powerrail
      Contact( "is_base_exsist" )
      wire#w1
      Contact( "state_of_start_base" )
      Contact( "is_base_exsist" )
      Coil( "base_raw_feeding_conveyr" )
   END_RUNG
   RUNG wire#powerrail
      Contact( "base_raw_feeding_conveyr" )
   END_RUNG wire#w1
   // the same network as SCL:
   "base_raw_feeding_conveyr" := ("is_base_exsist" OR "base_raw_feeding_conveyr") AND "state_of_start_base" AND "is_base_exsist";
END_REGION

REGION Network 7: base_machinning_handle
   RUNG wire#powerrail
      Contact( "is_base_exsist" )
      wire#w1
      Contact( "state_of_start_base" )
      Contact( "is_base_exsist" )
      Coil( "base_to_machinning_conveyr" )
   END_RUNG
   RUNG wire#powerrail
      Contact( "base_to_machinning_conveyr" )
   END_RUNG wire#w1
   // the same network as SCL:
   "base_to_machinning_conveyr" := ("is_base_exsist" OR "base_to_machinning_conveyr") AND "state_of_start_base" AND "is_base_exsist";
END_REGION

REGION Network 8: base_raw_into_cnc
   "IEC_Timer_0_DB_8".TOF(IN := NOT "base_into_cnc", PT := T#500ms);
   "is_base_exsist" := "IEC_Timer_0_DB_8".Q;
END_REGION

REGION Network 9: BASE_KEEP_DISTANCE
   RUNG wire#powerrail
      I_Contact( "is_base_exsist" )
      Coil( "Stop_blade4" )
      Coil( "Stop_blade5" )
   END_RUNG
   // the same network as SCL:
   "Stop_blade4" := NOT "is_base_exsist";
   "Stop_blade5" := NOT "is_base_exsist";
END_REGION

REGION Network 10: base_excess
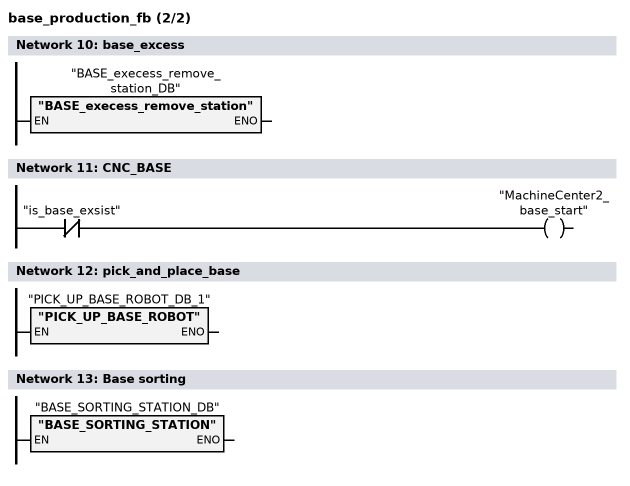
   RUNG wire#powerrail
      "BASE_execess_remove_station_DB"()
   END_RUNG
   // the same network as SCL:
   "BASE_execess_remove_station_DB"();   // "BASE_execess_remove_station"
END_REGION

REGION Network 11: CNC_BASE
   RUNG wire#powerrail
      I_Contact( "is_base_exsist" )
      Coil( "MachineCenter2_base_start" )
   END_RUNG
   // the same network as SCL:
   "MachineCenter2_base_start" := NOT "is_base_exsist";
END_REGION

REGION Network 12: pick_and_place_base
   RUNG wire#powerrail
      "PICK_UP_BASE_ROBOT_DB_1"()
   END_RUNG
   // the same network as SCL:
   "PICK_UP_BASE_ROBOT_DB_1"();   // "PICK_UP_BASE_ROBOT"
END_REGION

REGION Network 13: Base sorting
   RUNG wire#powerrail
      "BASE_SORTING_STATION_DB"()
   END_RUNG
   // the same network as SCL:
   "BASE_SORTING_STATION_DB"();   // "BASE_SORTING_STATION"
END_REGION
END_FUNCTION_BLOCK

FUNCTION_BLOCK "PICK_UP_BASE_ROBOT"   // FB6, LAD
{ S7_Optimized_Access := 'FALSE' }
VERSION : 0.1
   VAR_TEMP   // added for the SCL form of the ladder/FBD networks
      _w1 : Bool;
   END_VAR
BEGIN

REGION Network 1: BASE_PICKUP_ROBOT_LOWERING_Z_AXIS
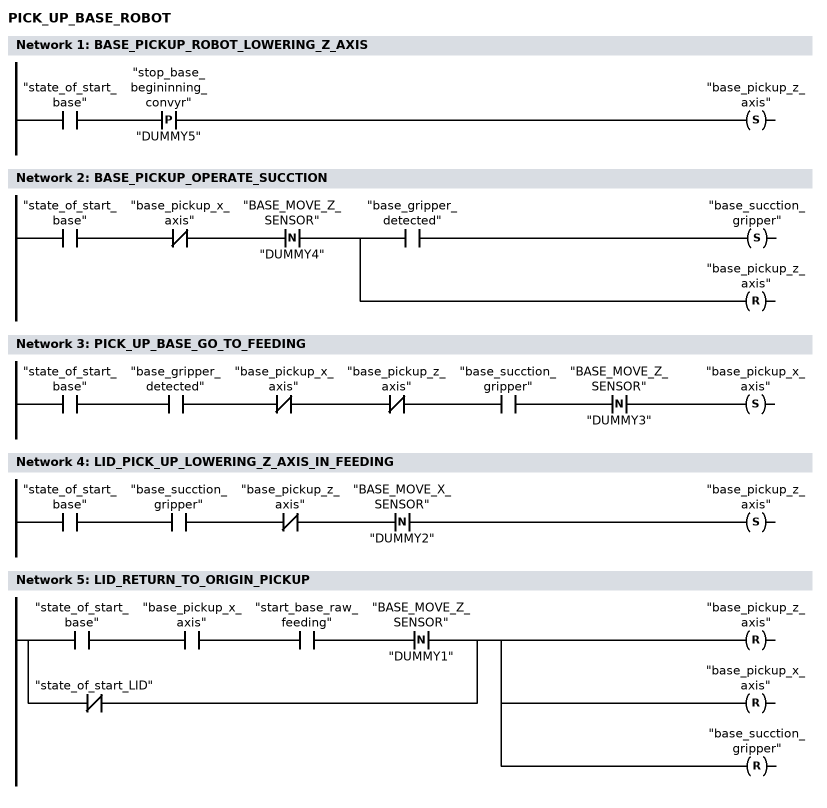
   RUNG wire#powerrail
      Contact( "state_of_start_base" )
      P_Contact(operand := "stop_base_begininning_convyr", bit := "DUMMY5")
      S_Coil( "base_pickup_z_axis" )
   END_RUNG
   // the same network as SCL:
   #_w1 := "state_of_start_base" AND "stop_base_begininning_convyr" AND NOT "DUMMY5";   // rising edge of "stop_base_begininning_convyr"
   "DUMMY5" := "stop_base_begininning_convyr";
   IF #_w1 THEN "base_pickup_z_axis" := TRUE; END_IF;
END_REGION

REGION Network 2: BASE_PICKUP_OPERATE_SUCCTION
   RUNG wire#powerrail
      Contact( "state_of_start_base" )
      I_Contact( "base_pickup_x_axis" )
      N_Contact(operand := "BASE_MOVE_Z_SENSOR", bit := "DUMMY4")
      wire#w1
      Contact( "base_gripper_detected" )
      S_Coil( "base_sucction_gripper" )
   END_RUNG
   RUNG wire#w1
      R_Coil( "base_pickup_z_axis" )
   END_RUNG
   // the same network as SCL:
   #_w1 := "state_of_start_base" AND NOT "base_pickup_x_axis" AND NOT "BASE_MOVE_Z_SENSOR" AND "DUMMY4";   // falling edge of "BASE_MOVE_Z_SENSOR"
   "DUMMY4" := "BASE_MOVE_Z_SENSOR";
   IF #_w1 AND "base_gripper_detected" THEN "base_sucction_gripper" := TRUE; END_IF;
   IF #_w1 THEN "base_pickup_z_axis" := FALSE; END_IF;
END_REGION

REGION Network 3: PICK_UP_BASE_GO_TO_FEEDING
   RUNG wire#powerrail
      Contact( "state_of_start_base" )
      Contact( "base_gripper_detected" )
      I_Contact( "base_pickup_x_axis" )
      I_Contact( "base_pickup_z_axis" )
      Contact( "base_sucction_gripper" )
      N_Contact(operand := "BASE_MOVE_Z_SENSOR", bit := "DUMMY3")
      S_Coil( "base_pickup_x_axis" )
   END_RUNG
   // the same network as SCL:
   #_w1 := "state_of_start_base" AND "base_gripper_detected" AND NOT "base_pickup_x_axis" AND NOT "base_pickup_z_axis" AND "base_sucction_gripper" AND NOT "BASE_MOVE_Z_SENSOR" AND "DUMMY3";   // falling edge of "BASE_MOVE_Z_SENSOR"
   "DUMMY3" := "BASE_MOVE_Z_SENSOR";
   IF #_w1 THEN "base_pickup_x_axis" := TRUE; END_IF;
END_REGION

REGION Network 4: LID_PICK_UP_LOWERING_Z_AXIS_IN_FEEDING
   RUNG wire#powerrail
      Contact( "state_of_start_base" )
      Contact( "base_sucction_gripper" )
      I_Contact( "base_pickup_z_axis" )
      N_Contact(operand := "BASE_MOVE_X_SENSOR", bit := "DUMMY2")
      S_Coil( "base_pickup_z_axis" )
   END_RUNG
   // the same network as SCL:
   #_w1 := "state_of_start_base" AND "base_sucction_gripper" AND NOT "base_pickup_z_axis" AND NOT "BASE_MOVE_X_SENSOR" AND "DUMMY2";   // falling edge of "BASE_MOVE_X_SENSOR"
   "DUMMY2" := "BASE_MOVE_X_SENSOR";
   IF #_w1 THEN "base_pickup_z_axis" := TRUE; END_IF;
END_REGION

REGION Network 5: LID_RETURN_TO_ORIGIN_PICKUP
   RUNG wire#powerrail
      Contact( "state_of_start_base" )
      Contact( "base_pickup_x_axis" )
      Contact( "start_base_raw_feeding" )
      N_Contact(operand := "BASE_MOVE_Z_SENSOR", bit := "DUMMY1")
      wire#w1
      R_Coil( "base_pickup_z_axis" )
   END_RUNG
   RUNG wire#powerrail
      I_Contact( "state_of_start_LID" )
   END_RUNG wire#w1
   RUNG wire#w1
      R_Coil( "base_pickup_x_axis" )
   END_RUNG
   RUNG wire#w1
      R_Coil( "base_sucction_gripper" )
   END_RUNG
   // the same network as SCL:
   #_w1 := "state_of_start_base" AND "base_pickup_x_axis" AND "start_base_raw_feeding" AND NOT "BASE_MOVE_Z_SENSOR" AND "DUMMY1";   // falling edge of "BASE_MOVE_Z_SENSOR"
   "DUMMY1" := "BASE_MOVE_Z_SENSOR";
   IF #_w1 OR NOT "state_of_start_LID" THEN
       "base_pickup_z_axis" := FALSE;
       "base_pickup_x_axis" := FALSE;
       "base_sucction_gripper" := FALSE;
   END_IF;
END_REGION
END_FUNCTION_BLOCK

FUNCTION_BLOCK "BASE_execess_remove_station"   // FB7, LAD
{ S7_Optimized_Access := 'FALSE' }
VERSION : 0.1
BEGIN

REGION Network 1: LID_BELT_EXECESS_CONVYR_HANDLER
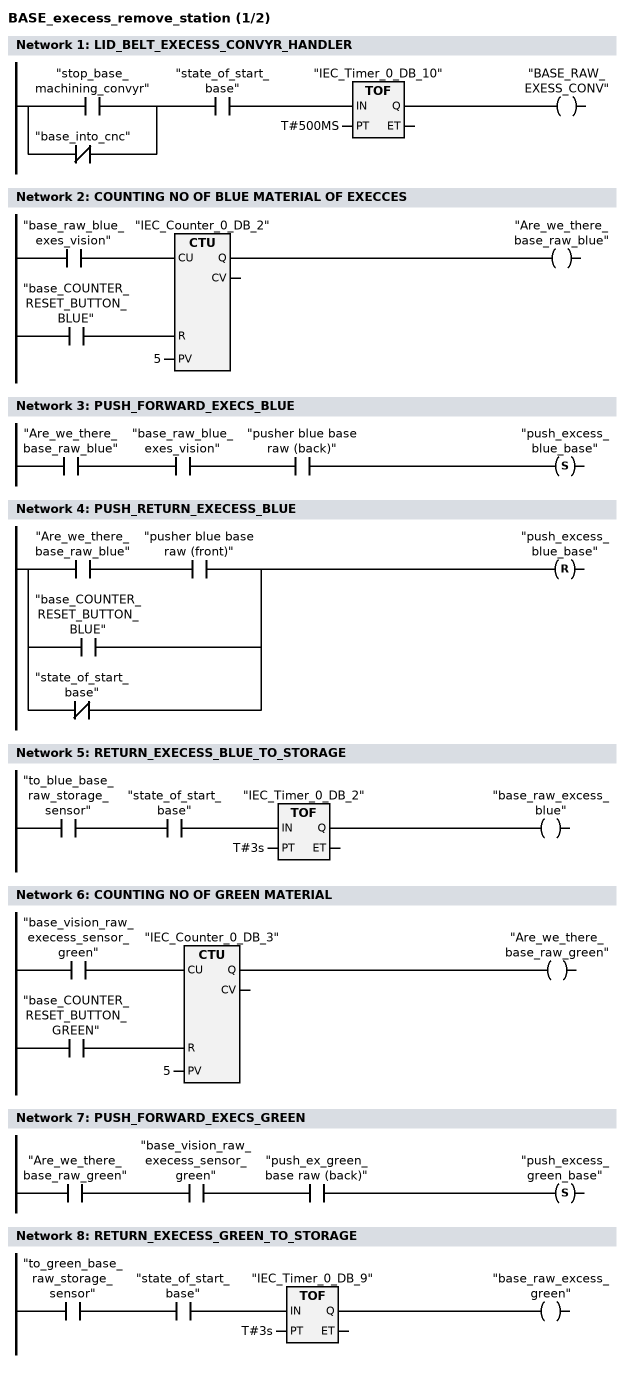
   "IEC_Timer_0_DB_10".TOF(IN := ("stop_base_machining_convyr" OR NOT "base_into_cnc") AND "state_of_start_base",
                           PT := T#500MS);
   "BASE_RAW_EXESS_CONV" := "IEC_Timer_0_DB_10".Q;
END_REGION

REGION Network 2: COUNTING NO OF BLUE MATERIAL OF EXECCES
   "IEC_Counter_0_DB_2".CTU(CU := "base_raw_blue_exes_vision", R := "base_COUNTER_RESET_BUTTON_BLUE", PV := 5);
   "Are_we_there_base_raw_blue" := "IEC_Counter_0_DB_2".Q;
END_REGION

REGION Network 3: PUSH_FORWARD_EXECS_BLUE
   RUNG wire#powerrail
      Contact( "Are_we_there_base_raw_blue" )
      Contact( "base_raw_blue_exes_vision" )
      Contact( "pusher blue base raw (back)" )
      S_Coil( "push_excess_blue_base" )
   END_RUNG
   // the same network as SCL:
   IF "Are_we_there_base_raw_blue" AND "base_raw_blue_exes_vision" AND "pusher blue base raw (back)" THEN
       "push_excess_blue_base" := TRUE;
   END_IF;
END_REGION

REGION Network 4: PUSH_RETURN_EXECESS_BLUE
   RUNG wire#powerrail
      Contact( "Are_we_there_base_raw_blue" )
      Contact( "pusher blue base raw (front)" )
      wire#w1
      R_Coil( "push_excess_blue_base" )
   END_RUNG
   RUNG wire#powerrail
      Contact( "base_COUNTER_RESET_BUTTON_BLUE" )
   END_RUNG wire#w1
   RUNG wire#powerrail
      I_Contact( "state_of_start_base" )
   END_RUNG wire#w1
   // the same network as SCL:
   IF ("Are_we_there_base_raw_blue" AND "pusher blue base raw (front)") OR "base_COUNTER_RESET_BUTTON_BLUE" OR NOT "state_of_start_base" THEN
       "push_excess_blue_base" := FALSE;
   END_IF;
END_REGION

REGION Network 5: RETURN_EXECESS_BLUE_TO_STORAGE
   "IEC_Timer_0_DB_2".TOF(IN := "to_blue_base_raw_storage_sensor" AND "state_of_start_base", PT := T#3s);
   "base_raw_excess_blue" := "IEC_Timer_0_DB_2".Q;
END_REGION

REGION Network 6: COUNTING NO OF GREEN MATERIAL
   "IEC_Counter_0_DB_3".CTU(CU := "base_vision_raw_execess_sensor_green",
                           R := "base_COUNTER_RESET_BUTTON_GREEN",
                           PV := 5);
   "Are_we_there_base_raw_green" := "IEC_Counter_0_DB_3".Q;
END_REGION

REGION Network 7: PUSH_FORWARD_EXECS_GREEN
   RUNG wire#powerrail
      Contact( "Are_we_there_base_raw_green" )
      Contact( "base_vision_raw_execess_sensor_green" )
      Contact( "push_ex_green_base raw (back)" )
      S_Coil( "push_excess_green_base" )
   END_RUNG
   // the same network as SCL:
   IF "Are_we_there_base_raw_green" AND "base_vision_raw_execess_sensor_green" AND "push_ex_green_base raw (back)" THEN
       "push_excess_green_base" := TRUE;
   END_IF;
END_REGION

REGION Network 8: RETURN_EXECESS_GREEN_TO_STORAGE
   "IEC_Timer_0_DB_9".TOF(IN := "to_green_base_raw_storage_sensor" AND "state_of_start_base", PT := T#3s);
   "base_raw_excess_green" := "IEC_Timer_0_DB_9".Q;
END_REGION

REGION Network 9: PUSH_RETURN_GREEN
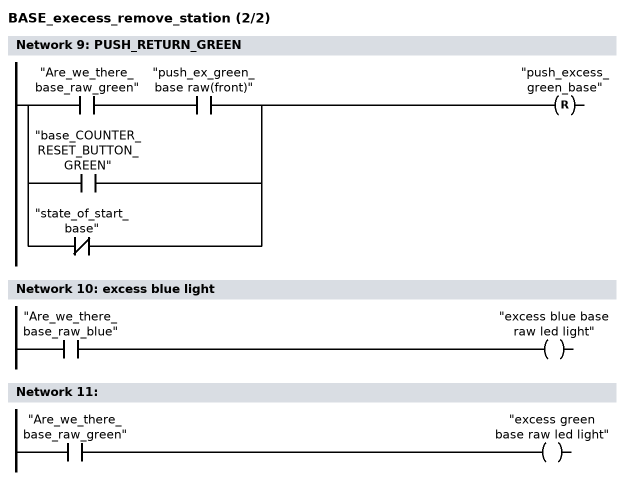
   RUNG wire#powerrail
      Contact( "Are_we_there_base_raw_green" )
      Contact( "push_ex_green_base raw(front)" )
      wire#w1
      R_Coil( "push_excess_green_base" )
   END_RUNG
   RUNG wire#powerrail
      Contact( "base_COUNTER_RESET_BUTTON_GREEN" )
   END_RUNG wire#w1
   RUNG wire#powerrail
      I_Contact( "state_of_start_base" )
   END_RUNG wire#w1
   // the same network as SCL:
   IF ("Are_we_there_base_raw_green" AND "push_ex_green_base raw(front)") OR "base_COUNTER_RESET_BUTTON_GREEN" OR NOT "state_of_start_base" THEN
       "push_excess_green_base" := FALSE;
   END_IF;
END_REGION

REGION Network 10: excess blue light
   RUNG wire#powerrail
      Contact( "Are_we_there_base_raw_blue" )
      Coil( "excess blue base raw led light" )
   END_RUNG
   // the same network as SCL:
   "excess blue base raw led light" := "Are_we_there_base_raw_blue";
END_REGION

REGION Network 11
   RUNG wire#powerrail
      Contact( "Are_we_there_base_raw_green" )
      Coil( "excess green base raw led light" )
   END_RUNG
   // the same network as SCL:
   "excess green base raw led light" := "Are_we_there_base_raw_green";
END_REGION
END_FUNCTION_BLOCK

FUNCTION_BLOCK "BASE_SORTING_STATION"   // FB8, LAD
{ S7_Optimized_Access := 'FALSE' }
VERSION : 0.1
BEGIN

REGION Network 1: BEGIN SORTING CONVYER
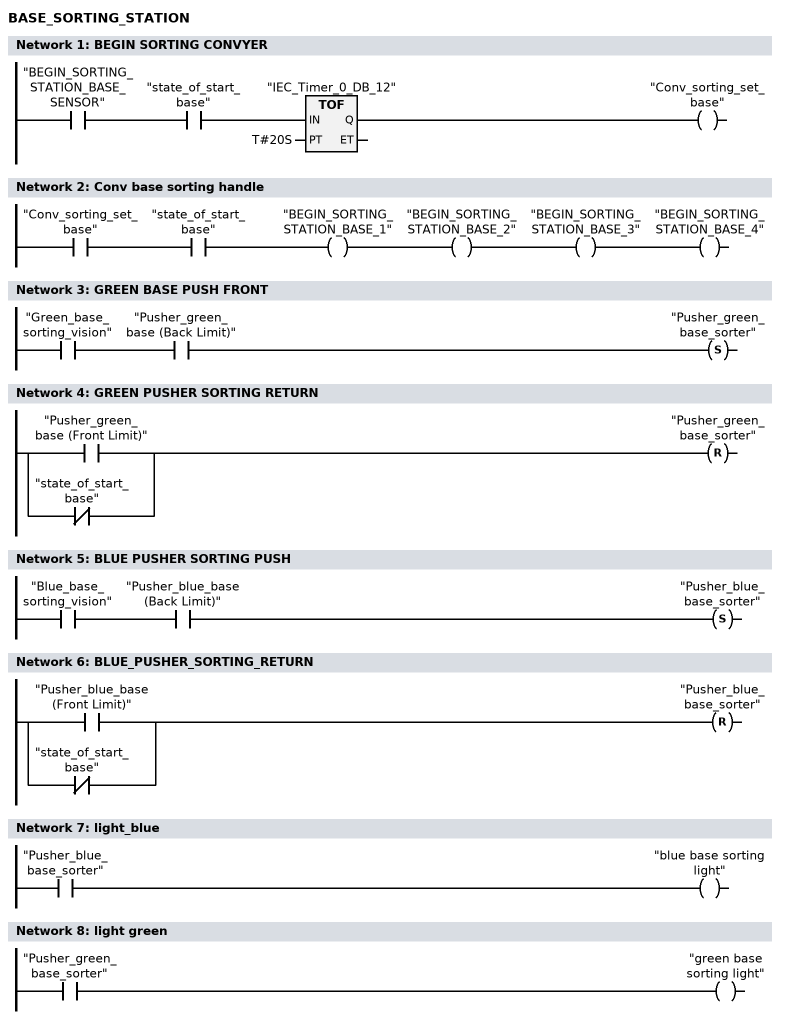
   "IEC_Timer_0_DB_12".TOF(IN := "BEGIN_SORTING_STATION_BASE_SENSOR" AND "state_of_start_base", PT := T#20S);
   "Conv_sorting_set_base" := "IEC_Timer_0_DB_12".Q;
END_REGION

REGION Network 2: Conv base sorting handle
   RUNG wire#powerrail
      Contact( "Conv_sorting_set_base" )
      Contact( "state_of_start_base" )
      Coil( "BEGIN_SORTING_STATION_BASE_1" )
      Coil( "BEGIN_SORTING_STATION_BASE_2" )
      Coil( "BEGIN_SORTING_STATION_BASE_3" )
      Coil( "BEGIN_SORTING_STATION_BASE_4" )
   END_RUNG
   // the same network as SCL:
   "BEGIN_SORTING_STATION_BASE_1" := "Conv_sorting_set_base" AND "state_of_start_base";
   "BEGIN_SORTING_STATION_BASE_2" := "BEGIN_SORTING_STATION_BASE_1";
   "BEGIN_SORTING_STATION_BASE_3" := "BEGIN_SORTING_STATION_BASE_1";
   "BEGIN_SORTING_STATION_BASE_4" := "BEGIN_SORTING_STATION_BASE_1";
END_REGION

REGION Network 3: GREEN BASE PUSH FRONT
   RUNG wire#powerrail
      Contact( "Green_base_sorting_vision" )
      Contact( "Pusher_green_base (Back Limit)" )
      S_Coil( "Pusher_green_base_sorter" )
   END_RUNG
   // the same network as SCL:
   IF "Green_base_sorting_vision" AND "Pusher_green_base (Back Limit)" THEN
       "Pusher_green_base_sorter" := TRUE;
   END_IF;
END_REGION

REGION Network 4: GREEN PUSHER SORTING RETURN
   RUNG wire#powerrail
      Contact( "Pusher_green_base (Front Limit)" )
      wire#w1
      R_Coil( "Pusher_green_base_sorter" )
   END_RUNG
   RUNG wire#powerrail
      I_Contact( "state_of_start_base" )
   END_RUNG wire#w1
   // the same network as SCL:
   IF "Pusher_green_base (Front Limit)" OR NOT "state_of_start_base" THEN
       "Pusher_green_base_sorter" := FALSE;
   END_IF;
END_REGION

REGION Network 5: BLUE PUSHER SORTING PUSH
   RUNG wire#powerrail
      Contact( "Blue_base_sorting_vision" )
      Contact( "Pusher_blue_base (Back Limit)" )
      S_Coil( "Pusher_blue_base_sorter" )
   END_RUNG
   // the same network as SCL:
   IF "Blue_base_sorting_vision" AND "Pusher_blue_base (Back Limit)" THEN
       "Pusher_blue_base_sorter" := TRUE;
   END_IF;
END_REGION

REGION Network 6: BLUE_PUSHER_SORTING_RETURN
   RUNG wire#powerrail
      Contact( "Pusher_blue_base (Front Limit)" )
      wire#w1
      R_Coil( "Pusher_blue_base_sorter" )
   END_RUNG
   RUNG wire#powerrail
      I_Contact( "state_of_start_base" )
   END_RUNG wire#w1
   // the same network as SCL:
   IF "Pusher_blue_base (Front Limit)" OR NOT "state_of_start_base" THEN
       "Pusher_blue_base_sorter" := FALSE;
   END_IF;
END_REGION

REGION Network 7: light_blue
   RUNG wire#powerrail
      Contact( "Pusher_blue_base_sorter" )
      Coil( "blue base sorting light" )
   END_RUNG
   // the same network as SCL:
   "blue base sorting light" := "Pusher_blue_base_sorter";
END_REGION

REGION Network 8: light green
   RUNG wire#powerrail
      Contact( "Pusher_green_base_sorter" )
      Coil( "green base sorting light" )
   END_RUNG
   // the same network as SCL:
   "green base sorting light" := "Pusher_green_base_sorter";
END_REGION
END_FUNCTION_BLOCK

FUNCTION_BLOCK "Assembly_conv"   // FB9, LAD
{ S7_Optimized_Access := 'FALSE' }
VERSION : 0.1
   VAR_TEMP   // added for the SCL form of the ladder/FBD networks
      _w1 : Bool;
      _s5time1 : S5Time;
   END_VAR
BEGIN

REGION Network 1
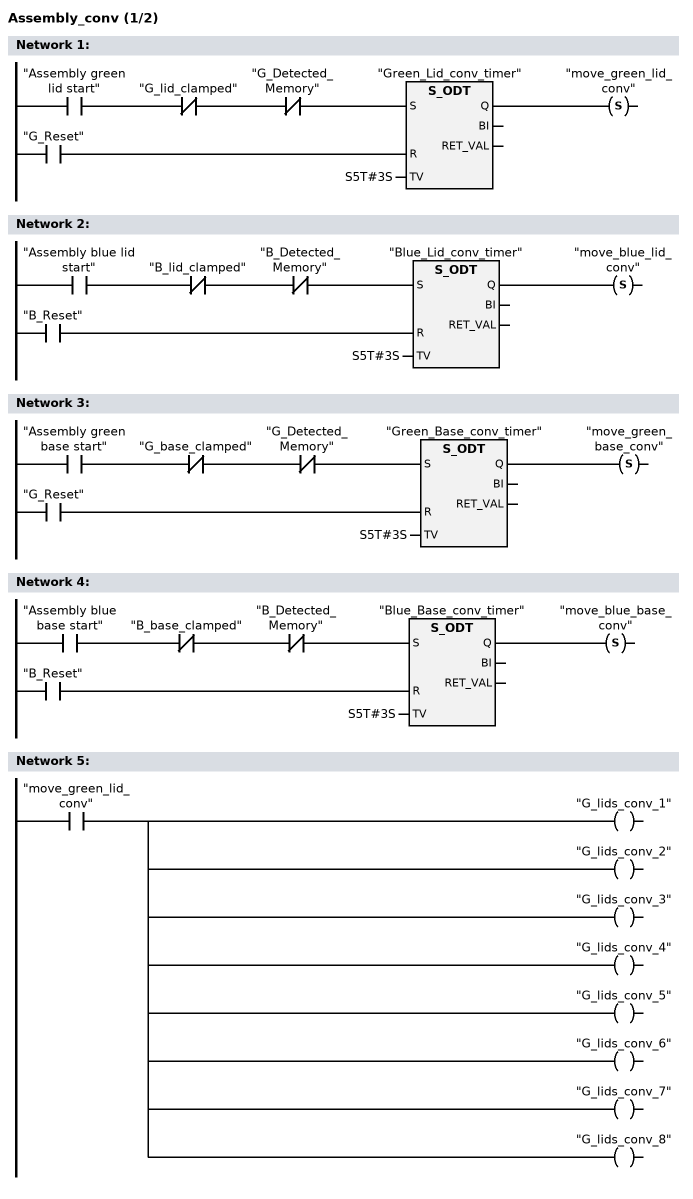
   RUNG wire#powerrail
      Contact( "Assembly green lid start" )
      I_Contact( "G_lid_clamped" )
      I_Contact( "G_Detected_Memory" )
      S_ODT(T_NO := "Green_Lid_conv_timer", R := wire#w1, TV := S5T#3S, BI =>, RET_VAL =>)
      S_Coil( "move_green_lid_conv" )
   END_RUNG
   RUNG wire#powerrail
      Contact( "G_Reset" )
   END_RUNG wire#w1
   // the same network as SCL:
   #_s5time1 := S_ODT(T_NO := "Green_Lid_conv_timer",
                      S := "Assembly green lid start" AND NOT "G_lid_clamped" AND NOT "G_Detected_Memory",
                      R := "G_Reset",
                      TV := S5T#3S,
                      Q => #_w1);
   IF #_w1 THEN "move_green_lid_conv" := TRUE; END_IF;
END_REGION

REGION Network 2
   RUNG wire#powerrail
      Contact( "Assembly blue lid start" )
      I_Contact( "B_lid_clamped" )
      I_Contact( "B_Detected_Memory" )
      S_ODT(T_NO := "Blue_Lid_conv_timer", R := wire#w1, TV := S5T#3S, BI =>, RET_VAL =>)
      S_Coil( "move_blue_lid_conv" )
   END_RUNG
   RUNG wire#powerrail
      Contact( "B_Reset" )
   END_RUNG wire#w1
   // the same network as SCL:
   #_s5time1 := S_ODT(T_NO := "Blue_Lid_conv_timer",
                      S := "Assembly blue lid start" AND NOT "B_lid_clamped" AND NOT "B_Detected_Memory",
                      R := "B_Reset",
                      TV := S5T#3S,
                      Q => #_w1);
   IF #_w1 THEN "move_blue_lid_conv" := TRUE; END_IF;
END_REGION

REGION Network 3
   RUNG wire#powerrail
      Contact( "Assembly green base start" )
      I_Contact( "G_base_clamped" )
      I_Contact( "G_Detected_Memory" )
      S_ODT(T_NO := "Green_Base_conv_timer", R := wire#w1, TV := S5T#3S, BI =>, RET_VAL =>)
      S_Coil( "move_green_base_conv" )
   END_RUNG
   RUNG wire#powerrail
      Contact( "G_Reset" )
   END_RUNG wire#w1
   // the same network as SCL:
   #_s5time1 := S_ODT(T_NO := "Green_Base_conv_timer",
                      S := "Assembly green base start" AND NOT "G_base_clamped" AND NOT "G_Detected_Memory",
                      R := "G_Reset",
                      TV := S5T#3S,
                      Q => #_w1);
   IF #_w1 THEN "move_green_base_conv" := TRUE; END_IF;
END_REGION

REGION Network 4
   RUNG wire#powerrail
      Contact( "Assembly blue base start" )
      I_Contact( "B_base_clamped" )
      I_Contact( "B_Detected_Memory" )
      S_ODT(T_NO := "Blue_Base_conv_timer", R := wire#w1, TV := S5T#3S, BI =>, RET_VAL =>)
      S_Coil( "move_blue_base_conv" )
   END_RUNG
   RUNG wire#powerrail
      Contact( "B_Reset" )
   END_RUNG wire#w1
   // the same network as SCL:
   #_s5time1 := S_ODT(T_NO := "Blue_Base_conv_timer",
                      S := "Assembly blue base start" AND NOT "B_base_clamped" AND NOT "B_Detected_Memory",
                      R := "B_Reset",
                      TV := S5T#3S,
                      Q => #_w1);
   IF #_w1 THEN "move_blue_base_conv" := TRUE; END_IF;
END_REGION

REGION Network 5
   RUNG wire#powerrail
      Contact( "move_green_lid_conv" )
      wire#w1
      Coil( "G_lids_conv_1" )
   END_RUNG
   RUNG wire#w1
      Coil( "G_lids_conv_2" )
   END_RUNG
   RUNG wire#w1
      Coil( "G_lids_conv_3" )
   END_RUNG
   RUNG wire#w1
      Coil( "G_lids_conv_4" )
   END_RUNG
   RUNG wire#w1
      Coil( "G_lids_conv_5" )
   END_RUNG
   RUNG wire#w1
      Coil( "G_lids_conv_6" )
   END_RUNG
   RUNG wire#w1
      Coil( "G_lids_conv_7" )
   END_RUNG
   RUNG wire#w1
      Coil( "G_lids_conv_8" )
   END_RUNG
   // the same network as SCL:
   "G_lids_conv_1" := "move_green_lid_conv";
   "G_lids_conv_2" := "move_green_lid_conv";
   "G_lids_conv_3" := "move_green_lid_conv";
   "G_lids_conv_4" := "move_green_lid_conv";
   "G_lids_conv_5" := "move_green_lid_conv";
   "G_lids_conv_6" := "move_green_lid_conv";
   "G_lids_conv_7" := "move_green_lid_conv";
   "G_lids_conv_8" := "move_green_lid_conv";
END_REGION

REGION Network 6
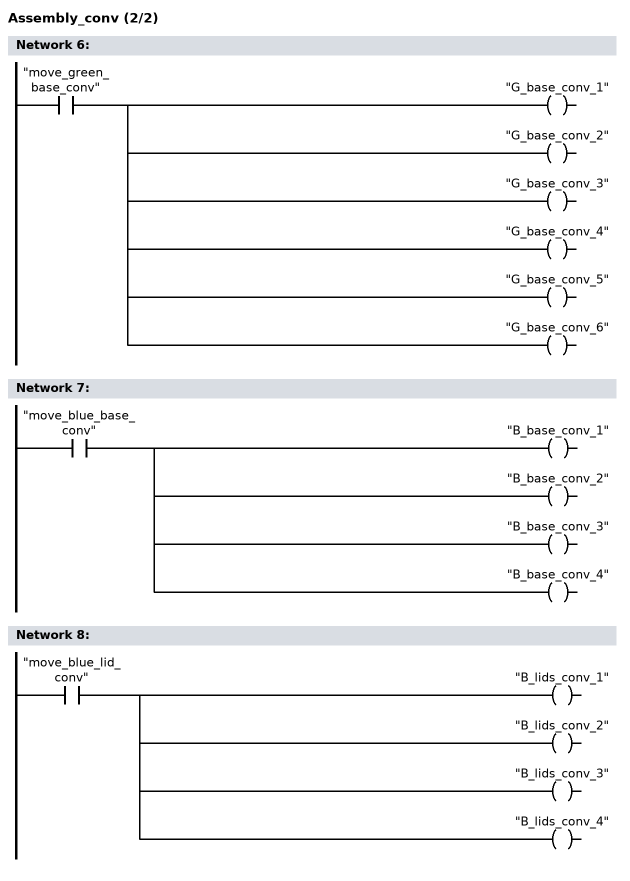
   RUNG wire#powerrail
      Contact( "move_green_base_conv" )
      wire#w1
      Coil( "G_base_conv_1" )
   END_RUNG
   RUNG wire#w1
      Coil( "G_base_conv_2" )
   END_RUNG
   RUNG wire#w1
      Coil( "G_base_conv_3" )
   END_RUNG
   RUNG wire#w1
      Coil( "G_base_conv_4" )
   END_RUNG
   RUNG wire#w1
      Coil( "G_base_conv_5" )
   END_RUNG
   RUNG wire#w1
      Coil( "G_base_conv_6" )
   END_RUNG
   // the same network as SCL:
   "G_base_conv_1" := "move_green_base_conv";
   "G_base_conv_2" := "move_green_base_conv";
   "G_base_conv_3" := "move_green_base_conv";
   "G_base_conv_4" := "move_green_base_conv";
   "G_base_conv_5" := "move_green_base_conv";
   "G_base_conv_6" := "move_green_base_conv";
END_REGION

REGION Network 7
   RUNG wire#powerrail
      Contact( "move_blue_base_conv" )
      wire#w1
      Coil( "B_base_conv_1" )
   END_RUNG
   RUNG wire#w1
      Coil( "B_base_conv_2" )
   END_RUNG
   RUNG wire#w1
      Coil( "B_base_conv_3" )
   END_RUNG
   RUNG wire#w1
      Coil( "B_base_conv_4" )
   END_RUNG
   // the same network as SCL:
   "B_base_conv_1" := "move_blue_base_conv";
   "B_base_conv_2" := "move_blue_base_conv";
   "B_base_conv_3" := "move_blue_base_conv";
   "B_base_conv_4" := "move_blue_base_conv";
END_REGION

REGION Network 8
   RUNG wire#powerrail
      Contact( "move_blue_lid_conv" )
      wire#w1
      Coil( "B_lids_conv_1" )
   END_RUNG
   RUNG wire#w1
      Coil( "B_lids_conv_2" )
   END_RUNG
   RUNG wire#w1
      Coil( "B_lids_conv_3" )
   END_RUNG
   RUNG wire#w1
      Coil( "B_lids_conv_4" )
   END_RUNG
   // the same network as SCL:
   "B_lids_conv_1" := "move_blue_lid_conv";
   "B_lids_conv_2" := "move_blue_lid_conv";
   "B_lids_conv_3" := "move_blue_lid_conv";
   "B_lids_conv_4" := "move_blue_lid_conv";
END_REGION
END_FUNCTION_BLOCK

FUNCTION_BLOCK "Assembly_Green"   // FB10, LAD
{ S7_Optimized_Access := 'FALSE' }
VERSION : 0.1
   VAR_TEMP   // added for the SCL form of the ladder/FBD networks
      _w1 : Bool;
      _s5time1 : S5Time;
   END_VAR
BEGIN

REGION Network 1
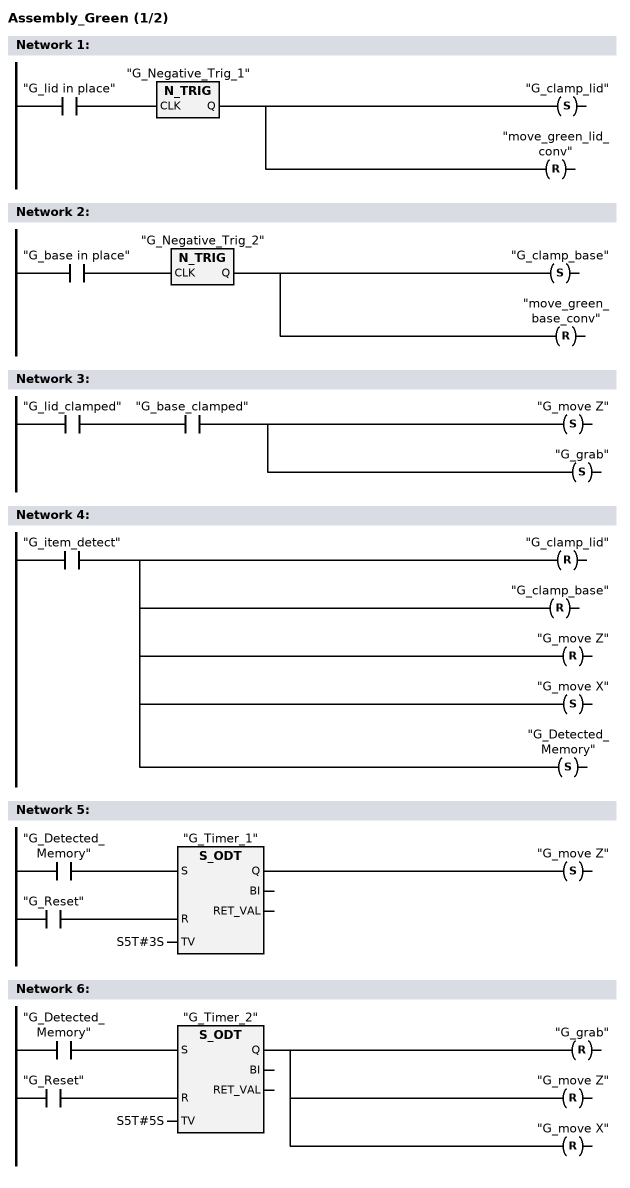
   RUNG wire#powerrail
      Contact( "G_lid in place" )
      N_Trig( "G_Negative_Trig_1" )
      wire#w1
      S_Coil( "G_clamp_lid" )
   END_RUNG
   RUNG wire#w1
      R_Coil( "move_green_lid_conv" )
   END_RUNG
   // the same network as SCL:
   #_w1 := NOT "G_lid in place" AND "G_Negative_Trig_1";   // falling edge
   "G_Negative_Trig_1" := "G_lid in place";
   IF #_w1 THEN
       "G_clamp_lid" := TRUE;
       "move_green_lid_conv" := FALSE;
   END_IF;
END_REGION

REGION Network 2
   RUNG wire#powerrail
      Contact( "G_base in place" )
      N_Trig( "G_Negative_Trig_2" )
      wire#w1
      S_Coil( "G_clamp_base" )
   END_RUNG
   RUNG wire#w1
      R_Coil( "move_green_base_conv" )
   END_RUNG
   // the same network as SCL:
   #_w1 := NOT "G_base in place" AND "G_Negative_Trig_2";   // falling edge
   "G_Negative_Trig_2" := "G_base in place";
   IF #_w1 THEN
       "G_clamp_base" := TRUE;
       "move_green_base_conv" := FALSE;
   END_IF;
END_REGION

REGION Network 3
   RUNG wire#powerrail
      Contact( "G_lid_clamped" )
      Contact( "G_base_clamped" )
      wire#w1
      S_Coil( "G_move Z" )
   END_RUNG
   RUNG wire#w1
      S_Coil( "G_grab" )
   END_RUNG
   // the same network as SCL:
   IF "G_lid_clamped" AND "G_base_clamped" THEN
       "G_move Z" := TRUE;
       "G_grab" := TRUE;
   END_IF;
END_REGION

REGION Network 4
   RUNG wire#powerrail
      Contact( "G_item_detect" )
      wire#w1
      R_Coil( "G_clamp_lid" )
   END_RUNG
   RUNG wire#w1
      R_Coil( "G_clamp_base" )
   END_RUNG
   RUNG wire#w1
      R_Coil( "G_move Z" )
   END_RUNG
   RUNG wire#w1
      S_Coil( "G_move X" )
   END_RUNG
   RUNG wire#w1
      S_Coil( "G_Detected_Memory" )
   END_RUNG
   // the same network as SCL:
   IF "G_item_detect" THEN
       "G_clamp_lid" := FALSE;
       "G_clamp_base" := FALSE;
       "G_move Z" := FALSE;
       "G_move X" := TRUE;
       "G_Detected_Memory" := TRUE;
   END_IF;
END_REGION

REGION Network 5
   RUNG wire#powerrail
      Contact( "G_Detected_Memory" )
      S_ODT(T_NO := "G_Timer_1", R := wire#w1, TV := S5T#3S, BI =>, RET_VAL =>)
      S_Coil( "G_move Z" )
   END_RUNG
   RUNG wire#powerrail
      Contact( "G_Reset" )
   END_RUNG wire#w1
   // the same network as SCL:
   #_s5time1 := S_ODT(T_NO := "G_Timer_1", S := "G_Detected_Memory", R := "G_Reset", TV := S5T#3S, Q => #_w1);
   IF #_w1 THEN "G_move Z" := TRUE; END_IF;
END_REGION

REGION Network 6
   RUNG wire#powerrail
      Contact( "G_Detected_Memory" )
      S_ODT(T_NO := "G_Timer_2", R := wire#w1, TV := S5T#5S, BI =>, RET_VAL =>)
      wire#w2
      R_Coil( "G_grab" )
   END_RUNG
   RUNG wire#powerrail
      Contact( "G_Reset" )
   END_RUNG wire#w1
   RUNG wire#w2
      R_Coil( "G_move Z" )
   END_RUNG
   RUNG wire#w2
      R_Coil( "G_move X" )
   END_RUNG
   // the same network as SCL:
   #_s5time1 := S_ODT(T_NO := "G_Timer_2", S := "G_Detected_Memory", R := "G_Reset", TV := S5T#5S, Q => #_w1);
   IF #_w1 THEN
       "G_grab" := FALSE;
       "G_move Z" := FALSE;
       "G_move X" := FALSE;
   END_IF;
END_REGION

REGION Network 7
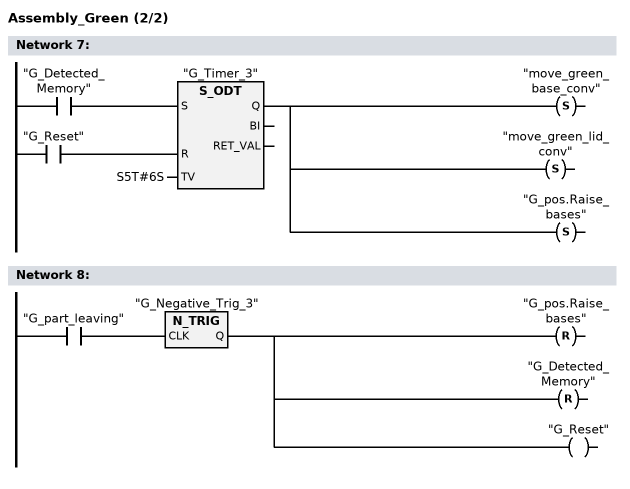
   RUNG wire#powerrail
      Contact( "G_Detected_Memory" )
      S_ODT(T_NO := "G_Timer_3", R := wire#w1, TV := S5T#6S, BI =>, RET_VAL =>)
      wire#w2
      S_Coil( "move_green_base_conv" )
   END_RUNG
   RUNG wire#powerrail
      Contact( "G_Reset" )
   END_RUNG wire#w1
   RUNG wire#w2
      S_Coil( "move_green_lid_conv" )
   END_RUNG
   RUNG wire#w2
      S_Coil( "G_pos.Raise_bases" )
   END_RUNG
   // the same network as SCL:
   #_s5time1 := S_ODT(T_NO := "G_Timer_3", S := "G_Detected_Memory", R := "G_Reset", TV := S5T#6S, Q => #_w1);
   IF #_w1 THEN
       "move_green_base_conv" := TRUE;
       "move_green_lid_conv" := TRUE;
       "G_pos.Raise_bases" := TRUE;
   END_IF;
END_REGION

REGION Network 8
   RUNG wire#powerrail
      Contact( "G_part_leaving" )
      N_Trig( "G_Negative_Trig_3" )
      wire#w1
      R_Coil( "G_pos.Raise_bases" )
   END_RUNG
   RUNG wire#w1
      R_Coil( "G_Detected_Memory" )
   END_RUNG
   RUNG wire#w1
      Coil( "G_Reset" )
   END_RUNG
   // the same network as SCL:
   #_w1 := NOT "G_part_leaving" AND "G_Negative_Trig_3";   // falling edge
   "G_Negative_Trig_3" := "G_part_leaving";
   IF #_w1 THEN
       "G_pos.Raise_bases" := FALSE;
       "G_Detected_Memory" := FALSE;
   END_IF;
   "G_Reset" := #_w1;
END_REGION
END_FUNCTION_BLOCK

FUNCTION_BLOCK "Assembly_Blue"   // FB11, LAD
{ S7_Optimized_Access := 'FALSE' }
VERSION : 0.1
   VAR_TEMP   // added for the SCL form of the ladder/FBD networks
      _w1 : Bool;
      _s5time1 : S5Time;
   END_VAR
BEGIN

REGION Network 1: Clamp when blue lid in place
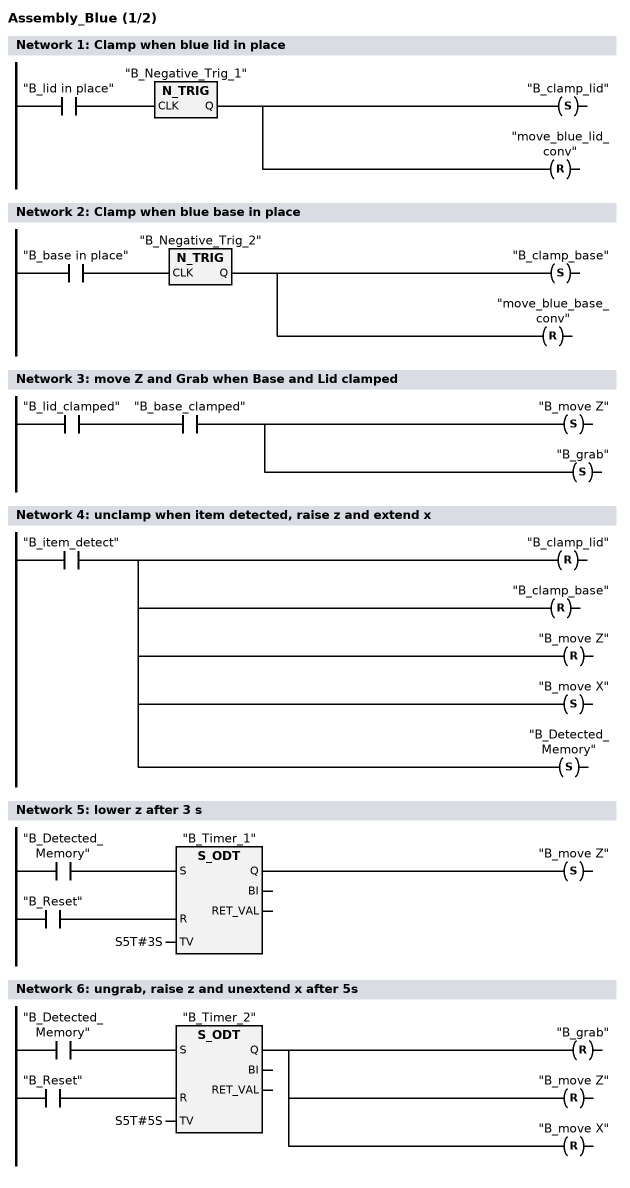
   RUNG wire#powerrail
      Contact( "B_lid in place" )
      N_Trig( "B_Negative_Trig_1" )
      wire#w1
      S_Coil( "B_clamp_lid" )
   END_RUNG
   RUNG wire#w1
      R_Coil( "move_blue_lid_conv" )
   END_RUNG
   // the same network as SCL:
   #_w1 := NOT "B_lid in place" AND "B_Negative_Trig_1";   // falling edge
   "B_Negative_Trig_1" := "B_lid in place";
   IF #_w1 THEN
       "B_clamp_lid" := TRUE;
       "move_blue_lid_conv" := FALSE;
   END_IF;
END_REGION

REGION Network 2: Clamp when blue base in place
   RUNG wire#powerrail
      Contact( "B_base in place" )
      N_Trig( "B_Negative_Trig_2" )
      wire#w1
      S_Coil( "B_clamp_base" )
   END_RUNG
   RUNG wire#w1
      R_Coil( "move_blue_base_conv" )
   END_RUNG
   // the same network as SCL:
   #_w1 := NOT "B_base in place" AND "B_Negative_Trig_2";   // falling edge
   "B_Negative_Trig_2" := "B_base in place";
   IF #_w1 THEN
       "B_clamp_base" := TRUE;
       "move_blue_base_conv" := FALSE;
   END_IF;
END_REGION

REGION Network 3: move Z and Grab when Base and Lid clamped
   RUNG wire#powerrail
      Contact( "B_lid_clamped" )
      Contact( "B_base_clamped" )
      wire#w1
      S_Coil( "B_move Z" )
   END_RUNG
   RUNG wire#w1
      S_Coil( "B_grab" )
   END_RUNG
   // the same network as SCL:
   IF "B_lid_clamped" AND "B_base_clamped" THEN
       "B_move Z" := TRUE;
       "B_grab" := TRUE;
   END_IF;
END_REGION

REGION Network 4: unclamp when item detected, raise z and extend x
   RUNG wire#powerrail
      Contact( "B_item_detect" )
      wire#w1
      R_Coil( "B_clamp_lid" )
   END_RUNG
   RUNG wire#w1
      R_Coil( "B_clamp_base" )
   END_RUNG
   RUNG wire#w1
      R_Coil( "B_move Z" )
   END_RUNG
   RUNG wire#w1
      S_Coil( "B_move X" )
   END_RUNG
   RUNG wire#w1
      S_Coil( "B_Detected_Memory" )
   END_RUNG
   // the same network as SCL:
   IF "B_item_detect" THEN
       "B_clamp_lid" := FALSE;
       "B_clamp_base" := FALSE;
       "B_move Z" := FALSE;
       "B_move X" := TRUE;
       "B_Detected_Memory" := TRUE;
   END_IF;
END_REGION

REGION Network 5: lower z after 3 s
   RUNG wire#powerrail
      Contact( "B_Detected_Memory" )
      S_ODT(T_NO := "B_Timer_1", R := wire#w1, TV := S5T#3S, BI =>, RET_VAL =>)
      S_Coil( "B_move Z" )
   END_RUNG
   RUNG wire#powerrail
      Contact( "B_Reset" )
   END_RUNG wire#w1
   // the same network as SCL:
   #_s5time1 := S_ODT(T_NO := "B_Timer_1", S := "B_Detected_Memory", R := "B_Reset", TV := S5T#3S, Q => #_w1);
   IF #_w1 THEN "B_move Z" := TRUE; END_IF;
END_REGION

REGION Network 6: ungrab, raise z and unextend x after 5s
   RUNG wire#powerrail
      Contact( "B_Detected_Memory" )
      S_ODT(T_NO := "B_Timer_2", R := wire#w1, TV := S5T#5S, BI =>, RET_VAL =>)
      wire#w2
      R_Coil( "B_grab" )
   END_RUNG
   RUNG wire#powerrail
      Contact( "B_Reset" )
   END_RUNG wire#w1
   RUNG wire#w2
      R_Coil( "B_move Z" )
   END_RUNG
   RUNG wire#w2
      R_Coil( "B_move X" )
   END_RUNG
   // the same network as SCL:
   #_s5time1 := S_ODT(T_NO := "B_Timer_2", S := "B_Detected_Memory", R := "B_Reset", TV := S5T#5S, Q => #_w1);
   IF #_w1 THEN
       "B_grab" := FALSE;
       "B_move Z" := FALSE;
       "B_move X" := FALSE;
   END_IF;
END_REGION

REGION Network 7: turn conv on and raise post after 6 s
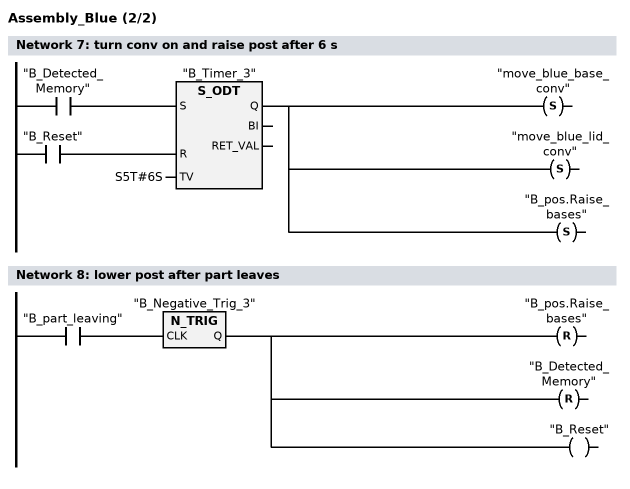
   RUNG wire#powerrail
      Contact( "B_Detected_Memory" )
      S_ODT(T_NO := "B_Timer_3", R := wire#w1, TV := S5T#6S, BI =>, RET_VAL =>)
      wire#w2
      S_Coil( "move_blue_base_conv" )
   END_RUNG
   RUNG wire#powerrail
      Contact( "B_Reset" )
   END_RUNG wire#w1
   RUNG wire#w2
      S_Coil( "move_blue_lid_conv" )
   END_RUNG
   RUNG wire#w2
      S_Coil( "B_pos.Raise_bases" )
   END_RUNG
   // the same network as SCL:
   #_s5time1 := S_ODT(T_NO := "B_Timer_3", S := "B_Detected_Memory", R := "B_Reset", TV := S5T#6S, Q => #_w1);
   IF #_w1 THEN
       "move_blue_base_conv" := TRUE;
       "move_blue_lid_conv" := TRUE;
       "B_pos.Raise_bases" := TRUE;
   END_IF;
END_REGION

REGION Network 8: lower post after part leaves
   RUNG wire#powerrail
      Contact( "B_part_leaving" )
      N_Trig( "B_Negative_Trig_3" )
      wire#w1
      R_Coil( "B_pos.Raise_bases" )
   END_RUNG
   RUNG wire#w1
      R_Coil( "B_Detected_Memory" )
   END_RUNG
   RUNG wire#w1
      Coil( "B_Reset" )
   END_RUNG
   // the same network as SCL:
   #_w1 := NOT "B_part_leaving" AND "B_Negative_Trig_3";   // falling edge
   "B_Negative_Trig_3" := "B_part_leaving";
   IF #_w1 THEN
       "B_pos.Raise_bases" := FALSE;
       "B_Detected_Memory" := FALSE;
   END_IF;
   "B_Reset" := #_w1;
END_REGION
END_FUNCTION_BLOCK

FUNCTION_BLOCK "A_COUNTER"   // FB12, LAD
{ S7_Optimized_Access := 'FALSE' }
VERSION : 0.1
BEGIN

REGION Network 1
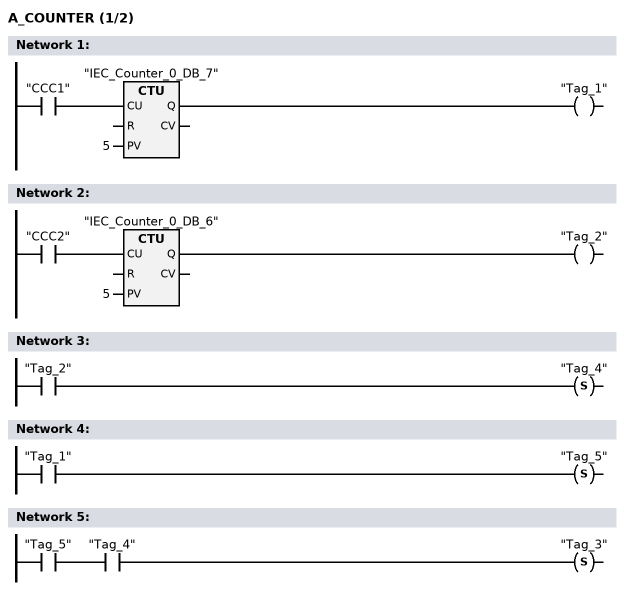
   "IEC_Counter_0_DB_7".CTU(CU := "CCC1", PV := 5);
   "Tag_1" := "IEC_Counter_0_DB_7".Q;
END_REGION

REGION Network 2
   "IEC_Counter_0_DB_6".CTU(CU := "CCC2", PV := 5);
   "Tag_2" := "IEC_Counter_0_DB_6".Q;
END_REGION

REGION Network 3
   RUNG wire#powerrail
      Contact( "Tag_2" )
      S_Coil( "Tag_4" )
   END_RUNG
   // the same network as SCL:
   IF "Tag_2" THEN "Tag_4" := TRUE; END_IF;
END_REGION

REGION Network 4
   RUNG wire#powerrail
      Contact( "Tag_1" )
      S_Coil( "Tag_5" )
   END_RUNG
   // the same network as SCL:
   IF "Tag_1" THEN "Tag_5" := TRUE; END_IF;
END_REGION

REGION Network 5
   RUNG wire#powerrail
      Contact( "Tag_5" )
      Contact( "Tag_4" )
      S_Coil( "Tag_3" )
   END_RUNG
   // the same network as SCL:
   IF "Tag_5" AND "Tag_4" THEN "Tag_3" := TRUE; END_IF;
END_REGION

REGION Network 6
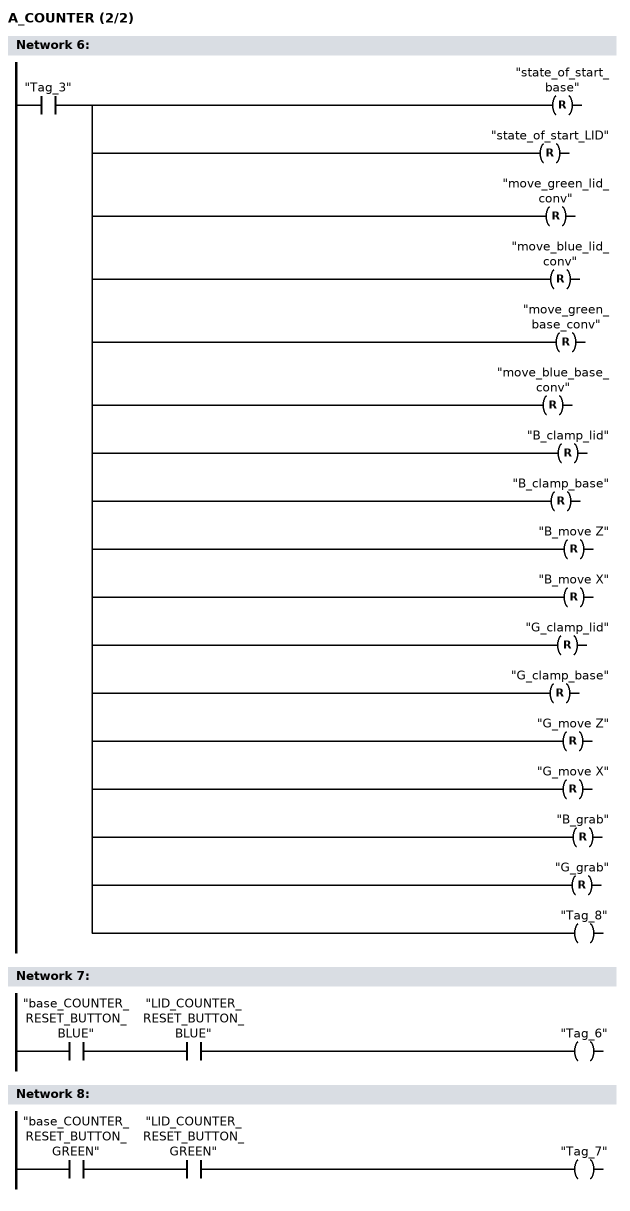
   RUNG wire#powerrail
      Contact( "Tag_3" )
      wire#w1
      R_Coil( "state_of_start_base" )
   END_RUNG
   RUNG wire#w1
      R_Coil( "state_of_start_LID" )
   END_RUNG
   RUNG wire#w1
      R_Coil( "move_green_lid_conv" )
   END_RUNG
   RUNG wire#w1
      R_Coil( "move_blue_lid_conv" )
   END_RUNG
   RUNG wire#w1
      R_Coil( "move_green_base_conv" )
   END_RUNG
   RUNG wire#w1
      R_Coil( "move_blue_base_conv" )
   END_RUNG
   RUNG wire#w1
      R_Coil( "B_clamp_lid" )
   END_RUNG
   RUNG wire#w1
      R_Coil( "B_clamp_base" )
   END_RUNG
   RUNG wire#w1
      R_Coil( "B_move Z" )
   END_RUNG
   RUNG wire#w1
      R_Coil( "B_move X" )
   END_RUNG
   RUNG wire#w1
      R_Coil( "G_clamp_lid" )
   END_RUNG
   RUNG wire#w1
      R_Coil( "G_clamp_base" )
   END_RUNG
   RUNG wire#w1
      R_Coil( "G_move Z" )
   END_RUNG
   RUNG wire#w1
      R_Coil( "G_move X" )
   END_RUNG
   RUNG wire#w1
      R_Coil( "B_grab" )
   END_RUNG
   RUNG wire#w1
      R_Coil( "G_grab" )
   END_RUNG
   RUNG wire#w1
      Coil( "Tag_8" )
   END_RUNG
   // the same network as SCL:
   IF "Tag_3" THEN
       "state_of_start_base" := FALSE;
       "state_of_start_LID" := FALSE;
       "move_green_lid_conv" := FALSE;
       "move_blue_lid_conv" := FALSE;
       "move_green_base_conv" := FALSE;
       "move_blue_base_conv" := FALSE;
       "B_clamp_lid" := FALSE;
       "B_clamp_base" := FALSE;
       "B_move Z" := FALSE;
       "B_move X" := FALSE;
       "G_clamp_lid" := FALSE;
       "G_clamp_base" := FALSE;
       "G_move Z" := FALSE;
       "G_move X" := FALSE;
       "B_grab" := FALSE;
       "G_grab" := FALSE;
   END_IF;
   "Tag_8" := "Tag_3";
END_REGION

REGION Network 7
   RUNG wire#powerrail
      Contact( "base_COUNTER_RESET_BUTTON_BLUE" )
      Contact( "LID_COUNTER_RESET_BUTTON_BLUE" )
      Coil( "Tag_6" )
   END_RUNG
   // the same network as SCL:
   "Tag_6" := "base_COUNTER_RESET_BUTTON_BLUE" AND "LID_COUNTER_RESET_BUTTON_BLUE";
END_REGION

REGION Network 8
   RUNG wire#powerrail
      Contact( "base_COUNTER_RESET_BUTTON_GREEN" )
      Contact( "LID_COUNTER_RESET_BUTTON_GREEN" )
      Coil( "Tag_7" )
   END_RUNG
   // the same network as SCL:
   "Tag_7" := "base_COUNTER_RESET_BUTTON_GREEN" AND "LID_COUNTER_RESET_BUTTON_GREEN";
END_REGION
END_FUNCTION_BLOCK

FUNCTION_BLOCK "Assembly_Emergency"   // FB13, LAD
{ S7_Optimized_Access := 'FALSE' }
VERSION : 0.1
BEGIN

REGION Network 1
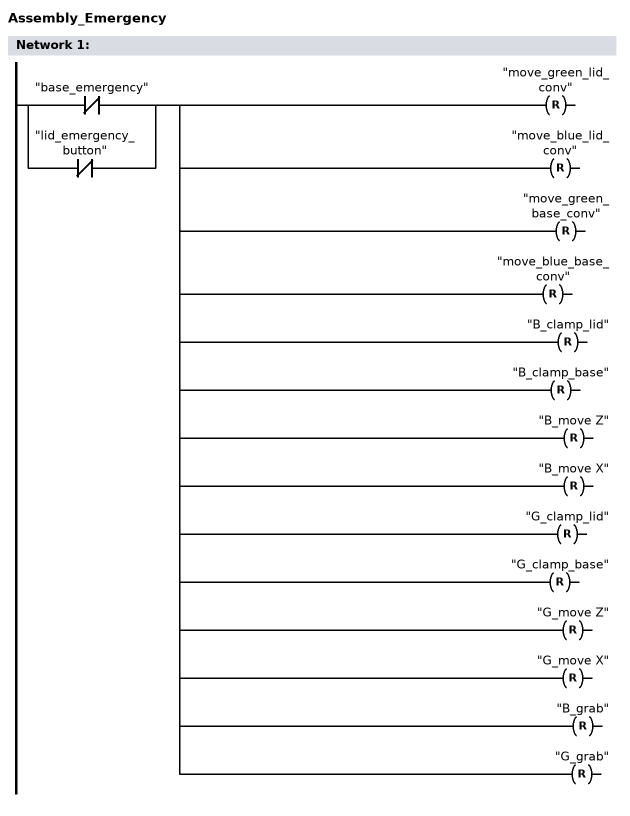
   RUNG wire#powerrail
      I_Contact( "base_emergency" )
      wire#w1
      R_Coil( "move_green_lid_conv" )
   END_RUNG
   RUNG wire#powerrail
      I_Contact( "lid_emergency_button" )
   END_RUNG wire#w1
   RUNG wire#w1
      R_Coil( "move_blue_lid_conv" )
   END_RUNG
   RUNG wire#w1
      R_Coil( "move_green_base_conv" )
   END_RUNG
   RUNG wire#w1
      R_Coil( "move_blue_base_conv" )
   END_RUNG
   RUNG wire#w1
      R_Coil( "B_clamp_lid" )
   END_RUNG
   RUNG wire#w1
      R_Coil( "B_clamp_base" )
   END_RUNG
   RUNG wire#w1
      R_Coil( "B_move Z" )
   END_RUNG
   RUNG wire#w1
      R_Coil( "B_move X" )
   END_RUNG
   RUNG wire#w1
      R_Coil( "G_clamp_lid" )
   END_RUNG
   RUNG wire#w1
      R_Coil( "G_clamp_base" )
   END_RUNG
   RUNG wire#w1
      R_Coil( "G_move Z" )
   END_RUNG
   RUNG wire#w1
      R_Coil( "G_move X" )
   END_RUNG
   RUNG wire#w1
      R_Coil( "B_grab" )
   END_RUNG
   RUNG wire#w1
      R_Coil( "G_grab" )
   END_RUNG
   // the same network as SCL:
   IF NOT "base_emergency" OR NOT "lid_emergency_button" THEN
       "move_green_lid_conv" := FALSE;
       "move_blue_lid_conv" := FALSE;
       "move_green_base_conv" := FALSE;
       "move_blue_base_conv" := FALSE;
       "B_clamp_lid" := FALSE;
       "B_clamp_base" := FALSE;
       "B_move Z" := FALSE;
       "B_move X" := FALSE;
       "G_clamp_lid" := FALSE;
       "G_clamp_base" := FALSE;
       "G_move Z" := FALSE;
       "G_move X" := FALSE;
       "B_grab" := FALSE;
       "G_grab" := FALSE;
   END_IF;
END_REGION
END_FUNCTION_BLOCK

ORGANIZATION_BLOCK "Main"   // OB1, LAD
TITLE = "Main Program Sweep (Cycle)"
{ S7_Optimized_Access := 'FALSE' }
VERSION : 0.1
   VAR_TEMP
      OB1_EV_CLASS : Byte;   // Bits 0-3 = 1 (Coming event), Bits 4-7 = 1 (Event class 1)
      OB1_SCAN_1 : Byte;   // 1 (Cold restart scan 1 of OB 1), 3 (Scan 2-n of OB 1)
      OB1_PRIORITY : Byte;   // Priority of OB Execution
      OB1_OB_NUMBR : Byte;   // 1 (Organization block 1, OB1)
      OB1_RESERVED_1 : Byte;   // Reserved for system
      OB1_RESERVED_2 : Byte;   // Reserved for system
      OB1_PREV_CYCLE : Int;   // Cycle time of previous OB1 scan (milliseconds)
      OB1_MIN_CYCLE : Int;   // Minimum cycle time of OB1 (milliseconds)
      OB1_MAX_CYCLE : Int;   // Maximum cycle time of OB1 (milliseconds)
      OB1_DATE_TIME : Date_And_Time;   // Date and time OB1 started
   END_VAR
BEGIN

REGION Network 1: LID_PRODUCTION_STATION
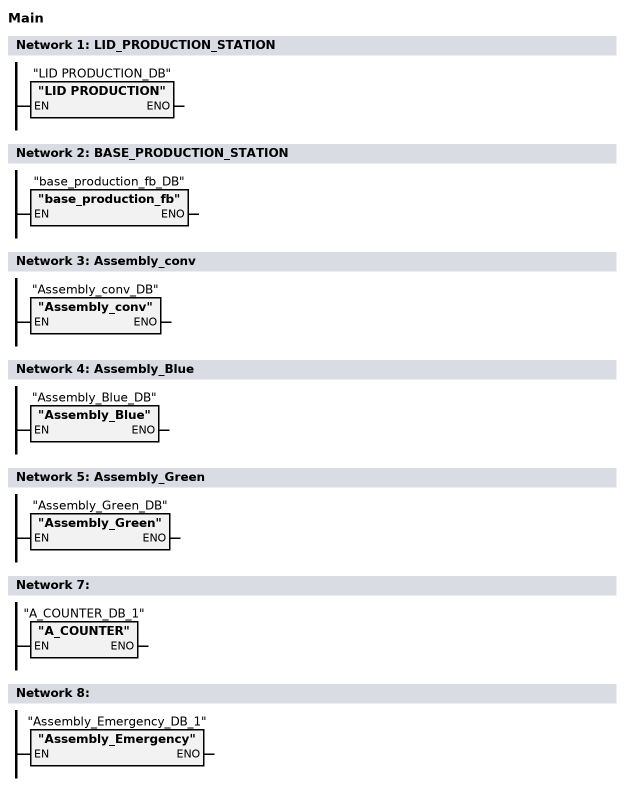
   RUNG wire#powerrail
      "LID PRODUCTION_DB"()
   END_RUNG
   // the same network as SCL:
   "LID PRODUCTION_DB"();   // "LID PRODUCTION"
END_REGION

REGION Network 2: BASE_PRODUCTION_STATION
   RUNG wire#powerrail
      "base_production_fb_DB"()
   END_RUNG
   // the same network as SCL:
   "base_production_fb_DB"();   // "base_production_fb"
END_REGION

REGION Network 3: Assembly_conv
   RUNG wire#powerrail
      "Assembly_conv_DB"()
   END_RUNG
   // the same network as SCL:
   "Assembly_conv_DB"();   // "Assembly_conv"
END_REGION

REGION Network 4: Assembly_Blue
   RUNG wire#powerrail
      "Assembly_Blue_DB"()
   END_RUNG
   // the same network as SCL:
   "Assembly_Blue_DB"();   // "Assembly_Blue"
END_REGION

REGION Network 5: Assembly_Green
   RUNG wire#powerrail
      "Assembly_Green_DB"()
   END_RUNG
   // the same network as SCL:
   "Assembly_Green_DB"();   // "Assembly_Green"
END_REGION

REGION Network 7
   RUNG wire#powerrail
      "A_COUNTER_DB_1"()
   END_RUNG
   // the same network as SCL:
   "A_COUNTER_DB_1"();   // "A_COUNTER"
END_REGION

REGION Network 8
   RUNG wire#powerrail
      "Assembly_Emergency_DB_1"()
   END_RUNG
   // the same network as SCL:
   "Assembly_Emergency_DB_1"();   // "Assembly_Emergency"
END_REGION
END_ORGANIZATION_BLOCK